(* IEC 61131-3 sources: SmartHomeNew/snapshots/2026-04-23, 16 files *)

(* ---- ST_Gateway_Command.dut ---- *)
{attribute 'pack_mode' := '1'}
TYPE ST_Gateway_Command :
STRUCT
    command_id : UDINT;
    timestamp_ms : UDINT;
    operator_id : STRING(10);
    command_type : E_Gateway_Command_Type;
    target_zone : BYTE;
    target_value : REAL;
    target_on_off : BOOL;
    target_scenario : E_SCENARIO_TYPE;
    target_armed : BOOL;
    target_pin : STRING(4);
    target_2fa_code : STRING(6);
    telegram_msg : STRING(200);
    source_ip : STRING(15); // IP-адрес источника команды для проверки безопасности
    crc32 : DWORD;
END_STRUCT
END_TYPE

(* ---- ST_Scenario_Config.dut ---- *)
{attribute 'pack_mode' := '1'}
TYPE ST_Scenario_Config :
STRUCT
    scenario_id : E_SCENARIO_TYPE;
    lighting_level_base : BYTE := 100;
    lighting_level_accent : BYTE := 100;
    floor_heating_adjust_celsius : REAL := 0.0;
    ventilation_speed_percent : BYTE := 50;
    sockets_enabled : BOOL := TRUE;
    blinds_position_percent : BYTE := 0;
    Presence_Simulation_Enabled : BOOL := FALSE;
END_STRUCT
END_TYPE

(* ---- ST_User_Rule.dut ---- *)
{attribute 'pack_mode' := '1'}
TYPE ST_User_Rule :
STRUCT
    Enabled : BOOL;
    Condition_Type : E_Rule_Condition_Type;
    Condition_Target_ID : BYTE; // ID зоны или датчика
    Condition_Op : E_Rule_Comparison;
    Condition_Value : REAL;
    Condition_Value_Max : REAL; // Для COMP_IN_RANGE
    Action_Target_ID : BYTE;
    Action_Value : REAL;
    Action_Type : E_Rule_Action_Type;
    Priority : BYTE;
END_STRUCT
END_TYPE

(* ---- GVL_CONFIG.gvl ---- *)
{attribute 'qualified_only'}
VAR_GLOBAL
    // Subsystem Configurations
    G_Heating_Config : ST_Heating_Config; // Настройки системы отопления
    G_Ventilation_Config : ST_Ventilation_Config; // Настройки системы вентиляции
    G_DHW_Config : ST_DHW_Config; // Настройки горячего водоснабжения
    G_Security_Config : ST_Security_Global_Config; // Настройки системы безопасности
    G_Flood_Config : ST_Flood_Config; // Настройки системы защиты от протечек

    // HMI Configurations
    G_HMI_FloorHeating_Configs : ARRAY[1..8] OF ST_FloorHeating_Circuit_Config; // Конфигурации контуров теплого пола
    G_Wet_Zone_Map : ARRAY[1..32] OF BOOL; // Карта мокрых зон (TRUE = мокрая зона)
    G_HMI_Tariff_Settings : ST_Tariff_Config; // Настройки тарифов
    G_HMI_Vent_Global_Config : ST_Ventilation_Global_Config; // Глобальные настройки вентиляции
    G_HMI_Vent_Unit_Configs : ARRAY[1..GVL_CONSTANTS.C_MAX_VENT_UNITS] OF ST_Ventilation_Unit_Config; // Конфигурации отдельных вентустановок
    G_HMI_Scenario_Configs : ARRAY[1..GVL_CONSTANTS.C_MAX_SCENARIOS] OF ST_Scenario_Config; // Конфигурации сценариев
    G_HMI_Outdoor_Configs : ARRAY[1..GVL_CONSTANTS.C_MAX_OUTDOOR_ZONES] OF ST_Outdoor_Zone_Config; // Конфигурации зон уличного освещения
    G_HMI_Flood_Config : ST_Flood_Global_Config; // Глобальные настройки защиты от протечек
    G_HMI_Gas_Config : ST_Gas_Valve_Configuration; // Конфигурация системы газового контроля
    G_HMI_Sensor_Calibrations : ARRAY[1..GVL_CONSTANTS.C_MAX_CALIBRATIONS] OF ST_Sensor_Calibration_Record; // Данные калибровки датчиков
    G_HMI_User_Rules : ARRAY[1..GVL_CONSTANTS.C_MAX_RULES] OF ST_User_Rule; // Пользовательские правила (Rule Engine)

    // Sensor calibration pipeline
    G_Enable_Sensor_Calibration : BOOL := TRUE;
    G_Calib_Outdoor_Temp : ST_Sensor_Calibration_Record;
    G_Calib_Supply_Temps : ARRAY[1..GVL_CONSTANTS.C_MAX_SUPPLY_TEMPS] OF ST_Sensor_Calibration_Record;
    G_Calib_Room_Temps : ARRAY[1..GVL_CONSTANTS.C_MAX_ZONES] OF ST_Sensor_Calibration_Record;
    G_Calib_Floor_Temps : ARRAY[1..GVL_CONSTANTS.C_MAX_ZONES] OF ST_Sensor_Calibration_Record;
    G_Calib_CO2 : ARRAY[1..GVL_CONSTANTS.C_MAX_ZONES] OF ST_Sensor_Calibration_Record;
    G_Calib_Humidity : ARRAY[1..GVL_CONSTANTS.C_MAX_ZONES] OF ST_Sensor_Calibration_Record;
    G_Calib_Manifold_T_Supply : ARRAY[1..GVL_CONSTANTS.C_MAX_MANIFOLDS] OF ST_Sensor_Calibration_Record;
    G_Calib_Manifold_T_Return : ARRAY[1..GVL_CONSTANTS.C_MAX_MANIFOLDS] OF ST_Sensor_Calibration_Record;
    G_Calib_Methane : ARRAY[1..GVL_CONSTANTS.C_MAX_METHANE_SENSORS] OF ST_Sensor_Calibration_Record;
    G_Calib_CO : ARRAY[1..GVL_CONSTANTS.C_MAX_CO_SENSORS] OF ST_Sensor_Calibration_Record;

    // Конфигурация тестирования клапанов
    G_Valve_Test_Config : ARRAY[1..GVL_CONSTANTS.C_MAX_MANIFOLDS] OF ST_Valve_Test_Config;

    // HMI Commands & States
    G_HMI_Cleaning_Mode_Active : ARRAY[1..GVL_CONSTANTS.C_MAX_CLEANING_MODES] OF BOOL; // Режим уборки активен
    G_HMI_Cleaning_Mode_TimeLeft : ARRAY[1..GVL_CONSTANTS.C_MAX_CLEANING_MODES] OF UINT; // Оставшееся время режима уборки
    G_HMI_Admin_2FA_Enabled : BOOL := FALSE; // Включена ли 2FA для ADMIN
    G_HMI_Current_Operator_Factor2_Done : BOOL; // Второй фактор пройден
    G_HMI_Current_Operator_ID : STRING(10); // ID текущего оператора
    G_HMI_Manual_Gas_Valve_Open : BOOL; // Ручное открытие газового клапана
    G_HMI_Manual_Gas_Valve_Time : UDINT := 5; // Время ручного открытия
    G_HMI_Manual_Gas_Valve_TimeLeft : UDINT; // Оставшееся время ручного открытия
    G_HMI_Apply_Settings : BOOL; // Команда: Применить настройки
    G_HMI_Mute_Alarm : BOOL; // Команда: Временное отключение сирены
    G_HMI_Ack_Alarms : BOOL; // Команда: Квитировать все тревоги

    // Access Control Commands
    G_HMI_Gate_Open_Req : BOOL; // Запрос на открытие въездных ворот
    G_HMI_Wicket_Open_Req : BOOL; // Запрос на открытие калитки
    G_HMI_Lock_1_Open_Req : BOOL; // Разблокировка основного замка
    G_HMI_Lock_1_Close_Req : BOOL; // Блокировка основного замка
    G_HMI_Lock_2_Open_Req : BOOL; // Разблокировка доп. замка
    G_HMI_Lock_2_Close_Req : BOOL; // Блокировка доп. замка

    // HMI Settings
    G_HMI_Language : BYTE := 0; // 0=RU, 1=EN
    G_HMI_Brightness : BYTE := 80;
    G_HMI_Screen_Saver_Timeout : UDINT := 300; // сек

    // Сетевая безопасность
    G_Allowed_IPs : ARRAY[1..GVL_CONSTANTS.C_MAX_ALLOWED_IPS] OF STRING(15) := ['192.168.1.100','192.168.1.101','127.0.0.1','','']; // Разрешенные IP-адреса для шлюза

    G_Backup_Circulation_Pump_In_Service : BOOL := TRUE; // Резервный насос доступен для логики
    G_Electric_Heater_In_Service : BOOL := TRUE; // Электронагреватель доступен для логики
    G_Freeze_Hardware_Retry_Count : INT := 2; // Количество повторных попыток для anti-freeze hardware
    G_Freeze_Hardware_Retry_Delay_MS : UDINT := 5000; // Задержка между попытками повторного пуска
    G_Pump_Exercise_Enabled : BOOL := TRUE; // Разрешение периодической прокрутки насосов после простоя
    G_Pump_Exercise_Interval_MS : UDINT := 604800000; // 7 суток
    G_Pump_Exercise_Duration_MS : UDINT := 30000; // 30 сек
    G_Manifold_Pump_In_Service : ARRAY[1..GVL_CONSTANTS.C_MAX_MANIFOLDS] OF BOOL := [TRUE, TRUE, TRUE, TRUE, TRUE];
    G_Manifold_Priority : ARRAY[1..GVL_CONSTANTS.C_MAX_MANIFOLDS] OF INT := [3, 3, 2, 2, 1]; // 3=high, 2=normal, 1=low
    G_Max_Active_Manifolds : INT := 3; // energy-management limit for simultaneous active manifolds
    G_Max_Thermal_Budget : REAL := 6.0; // simplified manifold thermal budget units
    G_DHW_Heating_Pump_In_Service : BOOL := TRUE;
    G_DHW_Circ_Pump_In_Service : BOOL := TRUE;
    G_Water_Valve_Exercise_Enabled : BOOL := TRUE;
    G_Water_Valve_Exercise_Interval_MS : UDINT := 604800000;
    G_Water_Valve_Exercise_Duration_MS : UDINT := 15000;
    G_Water_Valve_Exercise_Window_Start : TOD := TOD#04:00;
    G_Water_Valve_Exercise_Window_End : TOD := TOD#05:00;
    G_Water_Valve_Close_Retry_Count : INT := 2;
    G_Water_Valve_Close_Retry_Delay_MS : UDINT := 3000;
    // IO Mapping
    G_FloorTemp_Map : ARRAY[1..8] OF INT := [1, 2, 3, 4, 5, 6, 7, 8];
    G_RoomTemp_Map : ARRAY[1..16] OF INT := [1, 2, 3, 4, 5, 6, 7, 8, 9, 10, 11, 12, 13, 14, 15, 16];
    G_Door_Map : ARRAY[1..GVL_CONSTANTS.C_MAX_DOOR_SENSORS] OF INT := [1, 2, 3, 4, 5, 6, 7, 8];
    G_Window_Map : ARRAY[1..16] OF INT := [9, 10, 11, 12, 13, 14, 15, 16, 17, 18, 19, 20, 21, 22, 23, 24];

    // Evacuation config
    C_MAX_LIGHT_ZONES : INT := 32; // fallback if not defined elsewhere
    G_Evac_Exit_Zones : ARRAY[1..32] OF BOOL; // зоны-выходы (TRUE = выход)
    G_Evac_Smoke_Zone_Map : ARRAY[1..GVL_CONSTANTS.C_MAX_SMOKE_SENSORS] OF INT; // Привязка дымовых датчиков к зонам эвакуации
    G_Evac_Leak_Zone_Map : ARRAY[1..GVL_CONSTANTS.C_MAX_FLOOD_SENSORS] OF INT; // Привязка датчиков протечки к зонам эвакуации
    G_Evac_Gas_Zone_Map : ARRAY[1..GVL_CONSTANTS.C_MAX_METHANE_SENSORS] OF INT; // Привязка газовых датчиков к зонам эвакуации
    G_Evac_Zone_Names : ARRAY[1..32] OF STRING(80); // Человекочитаемые имена зон (помещения/крыло/этаж/сторона)

END_VAR

VAR_GLOBAL CONSTANT
    C_MS_PER_SEC    : UDINT := GVL_CONSTANTS.C_MS_IN_SECOND; // Миллисекунд в секунде
    C_SEC_PER_MIN   : UDINT := 60; // Секунд в минуте
    C_MIN_PER_HOUR  : UDINT := 60; // Минут в часе
    C_MS_PER_MIN    : UDINT := GVL_CONSTANTS.C_MS_IN_MINUTE; // Миллисекунд в минуте
    C_MAX_RULES     : INT := 20; // Максимальное количество пользовательских правил
    C_ZONE_COUNT    : BYTE := 18; // Общее количество зон в системе

    // Коды ошибок
    ERR_PRESSURE_OUT_OF_RANGE : UDINT := 16#E004;
    ERR_HIGH_DELTA_T : UDINT := 16#E005;
    ERR_BOILER_OFFLINE : UDINT := 16#E006;
    ERR_BOILER_GENERAL_FAULT : UDINT := 16#E007;
    ERR_BOILER_NO_FLAME : UDINT := 16#E008;
    ERR_PUMP_NO_CURRENT : UDINT := 16#E009;
    ERR_PUMP_UNDERCURRENT : UDINT := 16#E00A;
    ERR_PUMP_OVERCURRENT : UDINT := 16#E00B;
    ERR_DELTA_T_LOW : UDINT := 16#E00C;
    ERR_DELTA_T_HIGH : UDINT := 16#E00D;
    ERR_DHW_IO_OFFLINE : UDINT := 16#E00E;
    ERR_DHW_TEMP_SENSOR_FAULT : UDINT := 16#E00F;
    ERR_DHW_PRESSURE_OUT_OF_RANGE : UDINT := 16#E010;
    ERR_DHW_PRESSURE_SENSOR_FAULT : UDINT := 16#E011;
END_VAR

(* ---- GVL_IO.gvl ---- *)
{attribute 'qualified_only'}
VAR_GLOBAL
    DI_Security_Open : ARRAY[1..GVL_CONSTANTS.C_MAX_SECURITY_SENSORS] OF BOOL; // Дискретные входы: Герконы (нормально-замкнутые контакты, TRUE = Открыто)
    DI_Security_Glass : ARRAY[1..GVL_CONSTANTS.C_MAX_SECURITY_SENSORS] OF BOOL; // Дискретные входы: Датчики разбития стекла (активный уровень - TRUE)
    DI_Security_2F_Group : BOOL; // Дискретный вход: Групповой шлейф безопасности 2-го этажа (общий сигнал)
    DI_Flood_Sensors : ARRAY[1..GVL_CONSTANTS.C_MAX_FLOOD_SENSORS] OF BOOL; // Дискретные входы: Датчики протечки воды (активный уровень - TRUE)
    DI_Manifold_End_Switches : ARRAY[1..GVL_CONSTANTS.C_MAX_MANIFOLDS] OF BOOL; // Дискретные входы: Концевые выключатели клапанов коллекторов
    AO_Manifold_Valves : ARRAY[1..GVL_CONSTANTS.C_MAX_MANIFOLDS] OF UINT; // Аналоговые выходы: Приводы клапанов (0-10В, 0-1000 ед. для Modbus)
    DO_Manifold_Pumps : ARRAY[1..GVL_CONSTANTS.C_MAX_MANIFOLDS] OF BOOL; // Дискретные выходы: Циркуляционные насосы коллекторных узлов (220В)
    AI_Manifold_Currents : ARRAY[1..GVL_CONSTANTS.C_MAX_MANIFOLDS] OF INT; // Аналоговые входы: Обратная связь по току потребления насосов (диагностика)
    AI_Manifold_Pressures : ARRAY[1..GVL_CONSTANTS.C_MAX_MANIFOLDS] OF INT; // Аналоговые входы: Давление теплоносителя в коллекторах (0-10 бар)
    AI_Manifold_Temps_Supply : ARRAY[1..GVL_CONSTANTS.C_MAX_MANIFOLDS] OF ST_Owen_Analog_Value; // Аналоговые входы: Температура подачи (структура со статусом)
    AI_Manifold_Temps_Return : ARRAY[1..GVL_CONSTANTS.C_MAX_MANIFOLDS] OF INT; // Аналоговые входы: Температура обратной линии (в 10-х долях градуса)
    AO_Supply_Fans : ARRAY[1..GVL_CONSTANTS.C_MAX_SUPPLY_FANS] OF UINT; // Аналоговые выходы: Скорость приточных вентиляторов (0-10В)
    AO_Exhaust_Fans : ARRAY[1..GVL_CONSTANTS.C_MAX_EXHAUST_FANS] OF UINT; // Аналоговые выходы: Скорость вытяжных вентиляторов (0-10В)
    AO_Lighting_Levels : ARRAY[1..GVL_CONSTANTS.C_MAX_ZONES] OF UINT; // Аналоговые выходы: диммирование освещения (0-1000 -> 0..100%)
    AO_Blinds_Positions : ARRAY[1..GVL_CONSTANTS.C_MAX_BLINDS] OF UINT; // Аналоговые выходы: позиционирование штор/жалюзи (0-1000 -> 0..100%)
    AI_Supply_Temps : ARRAY[1..GVL_CONSTANTS.C_MAX_SUPPLY_TEMPS] OF ST_Owen_Analog_Value; // Аналоговые входы: Температура приточного воздуха после калорифера
    AI_Boiler_Modulation : ARRAY[1..GVL_CONSTANTS.C_MAX_BOILERS] OF INT; // Аналоговые входы: Текущий уровень модуляции мощности котла (%)
    AI_Boiler_Flame_Status : ARRAY[1..GVL_CONSTANTS.C_MAX_BOILERS] OF BOOL; // Дискретные входы: Датчик ионизации (подтверждение наличия пламени)
    DI_Boiler_Error : ARRAY[1..GVL_CONSTANTS.C_MAX_BOILERS] OF BOOL; // Дискретные входы: Сигнал общей ошибки/аварии котла
    AI_Methane_LEL : ARRAY[1..GVL_CONSTANTS.C_MAX_METHANE_SENSORS] OF ST_Owen_Analog_Value; // Аналоговые входы: Уровень метана CH4 (0-100% LEL)
    AI_CO_PPM : ARRAY[1..GVL_CONSTANTS.C_MAX_CO_SENSORS] OF REAL; // Аналоговые входы: Уровень угарного газа CO (PPM)
    DI_Smoke_Sensors : ARRAY[1..GVL_CONSTANTS.C_MAX_SMOKE_SENSORS] OF BOOL; // Дискретные входы: Оптические датчики дыма (пожарный шлейф)
    AI_Temp_Outdoor : ST_Owen_Analog_Value; // Аналоговый вход: Наружная температура воздуха (уличный датчик)
    AI_Floor_Temps : ARRAY[1..GVL_CONSTANTS.C_MAX_ZONES] OF REAL; // Аналоговые входы: Температура стяжки пола по зонам (датчики в гильзах)
    AI_Room_Temps : ARRAY[1..GVL_CONSTANTS.C_MAX_ZONES] OF REAL; // Аналоговые входы: Температура воздуха в помещениях (настенные датчики)
    AI_Room_Hum : ARRAY[1..GVL_CONSTANTS.C_MAX_ZONES] OF REAL; // Аналоговые входы: Влажность воздуха в помещениях (%)
    AI_Room_CO2 : ARRAY[1..GVL_CONSTANTS.C_MAX_ZONES] OF REAL; // Аналоговые входы: Уровень CO2 в помещениях (ppm)
    DO_Zone_Valves : ARRAY[1..GVL_CONSTANTS.C_MAX_ZONES] OF BOOL; // Дискретные выходы: Термоэлектрические приводы контуров (220В)
    AI_DHW_Temp : REAL; // Аналоговый вход: Температура воды в бойлере косвенного нагрева
    AI_DHW_Pressure : REAL; // Аналоговый вход: Давление в контуре ГВС (контроль подпитки и утечек)
    DO_DHW_Heating_Pump : BOOL; // Дискретный выход: Насос загрузки бойлера (первичный контур от котла)
    DO_DHW_Circ_Pump : BOOL; // Дискретный выход: Насос рециркуляции ГВС (кольцо потребителей)
    DO_Backup_Circulation_Pump : BOOL; // Дискретный выход: Резервный циркуляционный насос антизамерзания
    DO_Electric_Heater_Enable : BOOL; // Дискретный выход: Сухой контакт электрического нагревателя антизамерзания
    DI_Lighting_Switches : ARRAY[1..GVL_CONSTANTS.C_MAX_ZONES] OF BOOL; // Дискретные входы: Физические кнопки/выключатели (импульсные)
    DI_Socket_Switches : ARRAY[1..GVL_CONSTANTS.C_MAX_SOCKETS] OF BOOL; // Legacy-вход: локальные выключатели розеток отключены концептуально
    DI_Motion_Sensors : ARRAY[1..GVL_CONSTANTS.C_MAX_ZONES] OF BOOL; // Дискретные входы: Датчики присутствия (PIR-сенсоры)
    DO_Sockets : ARRAY[1..GVL_CONSTANTS.C_MAX_SOCKETS] OF BOOL; // Дискретные выходы: Управление розетками (реле)
    DO_Gas_Valve_Close : BOOL; // Дискретный выход: Импульс на закрытие электромагнитного газового клапана
    DO_Water_Valve_35_Close : BOOL; // Дискретный выход: Закрыть вводной шаровый кран воды №1 (с электроприводом)
    DO_Water_Valve_36_Close : BOOL; // Дискретный выход: Закрыть вводной шаровый кран воды №2 (с электроприводом)
    AI_Water_Valve_35_Current : REAL; // Аналоговый вход: Ток потребления электропривода крана №1 (контроль заклинивания)
    AI_Water_Valve_36_Current : REAL; // Аналоговый вход: Ток потребления электропривода крана №2 (контроль заклинивания)
    DI_Power_OK : BOOL; // Дискретный вход: Контроль наличия напряжения на вводе (реле контроля фаз)
    DO_Gas_Siren : BOOL; // Дискретный выход: Звуковое оповещение при опасной концентрации газа
    DO_Fire_Siren : BOOL; // Дискретный выход: Звуковое оповещение при обнаружении задымления
    DO_Security_Siren : BOOL; // Дискретный выход: Сирена охранной сигнализации
    DO_Pump_Main_Enable : BOOL; // Дискретный выход: Разрешение работы главного циркуляционного насоса системы
    DO_Gate_Open : BOOL; // Дискретный выход: Команда на открытие въездных ворот (импульс)
    DO_Wicket_Open : BOOL; // Дискретный выход: Команда на разблокировку электрозамка калитки
    DO_Lock_1_Open : BOOL; // Дискретный выход: Разблокировать основной электромеханический замок дома
    DO_Lock_1_Close : BOOL; // Дискретный выход: Заблокировать основной электромеханический замок дома
    DO_Lock_2_Open : BOOL; // Дискретный выход: Разблокировать дополнительный замок (черный ход)
    DO_Lock_2_Close : BOOL; // Дискретный выход: Заблокировать дополнительный замок (черный ход)
    DI_Partner_Pulse : BOOL; // Дискретный вход: Пульс от второго ПЛК
    DI_Partner_Active : BOOL; // Дискретный вход: Статус активности второго ПЛК
    DO_Heartbeat_Pulse : BOOL; // Дискретный выход: Собственный пульс
    DO_Active_Status : BOOL; // Дискретный выход: Собственный статус активности

    // Диагностика модулей ввода-вывода
    DI_Module_1_Heartbeat : BOOL; // Сигнал жизни от модуля 1
    DI_Module_2_Heartbeat : BOOL; // Сигнал жизни от модуля 2
    DI_Backup_Circulation_Pump_Feedback : BOOL; // Обратная связь резервного циркуляционного насоса
    DI_Electric_Heater_Feedback : BOOL; // Обратная связь электрического нагревателя
    DI_Water_Zone_Open_FB : ARRAY[1..32] OF BOOL; // Концевики: зональный водяной клапан открыт
    DI_Water_Zone_Close_FB : ARRAY[1..32] OF BOOL; // Концевики: зональный водяной клапан закрыт
    DO_Water_Zone_Enable : ARRAY[1..32] OF BOOL; // Разрешение подачи воды по зонам
END_VAR

(* ---- GVL_STATUS.gvl ---- *)
{attribute 'qualified_only'}
VAR_GLOBAL
    G_System_Time_MS : UDINT; // Системное время в миллисекундах
    G_Last_System_Time_MS : UDINT := 0; // Предыдущее системное время (для детекции переполнения)
    G_Time_Of_Day_MS : UDINT := 0; // Время от начала суток в мс (0-86399999)
    G_Current_Day : UINT := 1; // Текущий день недели (1-7)
    G_Day_Of_Year : UINT := 1; // Текущий день года (1-365)
    G_Current_TOD : TOD; // Текущее время суток
    G_Current_Scenario : E_SCENARIO_TYPE := E_SCENARIO_TYPE.SCENARIO_NONE; // Текущий активный сценарий
    G_Previous_Scenario : E_SCENARIO_TYPE := E_SCENARIO_TYPE.SCENARIO_NONE; // Предыдущий сценарий
    G_Is_Night : BOOL; // Флаг ночного времени
    G_PLC_ID : BYTE := 1; // 1 = PLC_A, 2 = PLC_B
    G_Is_Active_PLC : BOOL;
    G_Local_PLC_ID : BYTE := 1; // Идентификатор данного ПЛК в паре
    G_Active_PLC_ID : BYTE := 1; // Идентификатор ведущего ПЛК
    G_Remote_PLC_Pulse : BOOL; // Сигнал "жизни" от второго ПЛК
    G_Security_Status_Msg : STRING(200);
    G_Gas_Status_Msg : STRING(200);
    G_Flood_Status_Msg : STRING(200);
    G_Vent_Status_Msg : STRING(200);
    G_DHW_Status : ST_DHW_Status;
    G_Manifold_Status : ARRAY[1..GVL_CONSTANTS.C_MAX_MANIFOLDS] OF ST_Manifold_Status;
    G_Boiler_Status : ARRAY[1..GVL_CONSTANTS.C_MAX_BOILERS] OF ST_Boiler_Status;
    G_IO_Modules_Online : ARRAY[1..GVL_CONSTANTS.C_MAX_MODULES] OF BOOL; // Статусы модулей ввода-вывода
    G_Sim_Active : BOOL;
    G_Wet_Zone_Light_Active : BOOL;
    G_System_Mode_Msg : STRING(200); // Пояснение текущего режима работы системы для HMI
    G_System_Mode_Cause : STRING(200); // Корневая причина режима (пожар/газ/протечка/штатно)
    G_Evac_Target_Zone_Name : STRING(80); // Предпочтительная зона выхода/направления эвакуации
    G_Evac_Hazard_Zone_Name : STRING(80); // Наиболее важная опасная зона для HMI/диагностики
    G_Diagnostics : ST_System_Diagnostics; // Интегральная диагностика и HMI-состояния
END_VAR

(* ---- FB_Access_Control.st ---- *)
FUNCTION_BLOCK FB_Access_Control
VAR_INPUT
    VI_System_Time_MS   : UDINT; // Системное время (мс)
    VI_IsActivePLC      : BOOL; // Флаг: Данный ПЛК является ведущим (Active)
    VI_Armed            : BOOL; // Статус: Система безопасности находится под охраной
    VI_System_Mode      : E_System_Operating_Mode; // Агрегированный режим работы системы

    // Команды управления от HMI (через GVL_CONFIG)
    VI_Gate_Open_Req    : BOOL; // Запрос пользователя на открытие въездных ворот
    VI_Wicket_Open_Req  : BOOL; // Запрос пользователя на открытие калитки
    VI_Lock_1_Open_Req  : BOOL; // Запрос на разблокировку основного электрозамка дома
    VI_Lock_1_Close_Req : BOOL; // Запрос на блокировку основного электрозамка дома
    VI_Lock_2_Open_Req  : BOOL; // Запрос на разблокировку дополнительного электрозамка
    VI_Lock_2_Close_Req : BOOL; // Запрос на блокировку дополнительного электрозамка

    // Авторизация
    VI_PIN_Code         : STRING(4); // ПИН-код для авторизации
    VI_RFID_Tag         : STRING(20); // RFID/NFC метка для авторизации

    // Настройки из конфигурации безопасности (длительности импульсов)
    VI_Config           : ST_Security_Global_Config;
END_VAR
VAR_IN_OUT
    VI_Access_Codes     : ARRAY[1..GVL_CONSTANTS.C_MAX_ACCESS_CODES] OF DWORD;
    VI_RFID_Tags        : ARRAY[1..GVL_CONSTANTS.C_MAX_ACCESS_CODES] OF STRING(20);
END_VAR
VAR_OUTPUT
    VO_Gate_Open        : BOOL; // Выход: Импульс на открытие ворот (сухой контакт)
    VO_Wicket_Open      : BOOL; // Выход: Импульс на открытие калитки (электрозащелка)
    VO_Lock_1_Open      : BOOL; // Выход: Импульс на разблокировку замка №1
    VO_Lock_1_Close     : BOOL; // Выход: Импульс на блокировку замка №1
    VO_Lock_2_Open      : BOOL; // Выход: Импульс на разблокировку замка №2
    VO_Lock_2_Close     : BOOL; // Выход: Импульс на блокировку замка №2
END_VAR
VAR
    // Таймеры для формирования импульсов управления заданной длительности
    L_Gate_Timer        : TP; // Таймер импульса ворот
    L_Wicket_Timer      : TP; // Таймер импульса калитки
    L_Lock_1_Open_T     : TP; // Таймер открытия замка №1
    L_Lock_1_Close_T    : TP; // Таймер закрытия замка №1
    L_Lock_2_Open_T     : TP; // Таймер открытия замка №2
    L_Lock_2_Close_T    : TP; // Таймер закрытия замка №2

    L_Prev_Armed        : BOOL; // Предыдущее состояние охраны (для детекции фронта постановки)
    L_Auto_Lock_Req     : BOOL; // Флаг автоматического закрытия всех замков при постановке на охрану

    R_Trig_Gate         : R_TRIG;
    R_Trig_Wicket       : R_TRIG;
    R_Trig_Lock_1_O     : R_TRIG;
    R_Trig_Lock_1_C     : R_TRIG;
    R_Trig_Lock_2_O     : R_TRIG;
    R_Trig_Lock_2_C     : R_TRIG;

    fbAccessCode        : FB_AccessCode_Manager;
    L_Valid_PIN         : BOOL;
END_VAR

// Если ПЛК находится в режиме Standby (резерв), он не должен управлять выходами
IF NOT VI_IsActivePLC THEN
    RETURN;
END_IF;

IF VI_System_Mode = E_System_Operating_Mode.MODE_SAFE_STOP THEN
    VO_Gate_Open := FALSE;
    VO_Wicket_Open := FALSE;
    VO_Lock_1_Open := FALSE;
    VO_Lock_2_Open := FALSE;
    RETURN;
END_IF;

// 1. Логика автоматического закрытия замков при постановке на охрану (ТЗ 3.0)
// При переходе системы в режим "Охрана" принудительно блокируем все замки
IF VI_Armed AND NOT L_Prev_Armed THEN
    L_Auto_Lock_Req := TRUE;
END_IF;
L_Prev_Armed := VI_Armed;

// Детекторы фронта для команд
R_Trig_Gate(CLK := VI_Gate_Open_Req);
R_Trig_Wicket(CLK := VI_Wicket_Open_Req);
R_Trig_Lock_1_O(CLK := VI_Lock_1_Open_Req);
R_Trig_Lock_1_C(CLK := VI_Lock_1_Close_Req OR L_Auto_Lock_Req);
R_Trig_Lock_2_O(CLK := VI_Lock_2_Open_Req);
R_Trig_Lock_2_C(CLK := VI_Lock_2_Close_Req OR L_Auto_Lock_Req);

// Проверка PIN-кода или RFID-метки через менеджер кодов
fbAccessCode(
    VI_System_Time_MS := VI_System_Time_MS,
    VI_IsActivePLC := VI_IsActivePLC,
    VI_Code_To_Check := VI_PIN_Code,
    VI_RFID_To_Check := VI_RFID_Tag,
    VI_Access_Codes := VI_Access_Codes,
    VI_RFID_Tags := VI_RFID_Tags,
    VO_Code_Valid => L_Valid_PIN
);

// 2. Формирование импульсов управления исполнительными механизмами (Pulse Control)
// Открытие ворот и калитки требует валидного ПИН-кода или RFID-метки, если система под охраной
L_Gate_Timer(IN := R_Trig_Gate.Q AND (NOT VI_Armed OR L_Valid_PIN), PT := TO_TIME(VI_Config.gate_open_pulse_ms));
VO_Gate_Open := L_Gate_Timer.Q;

L_Wicket_Timer(IN := R_Trig_Wicket.Q AND (NOT VI_Armed OR L_Valid_PIN), PT := TO_TIME(VI_Config.wicket_open_pulse_ms));
VO_Wicket_Open := L_Wicket_Timer.Q;

L_Lock_1_Open_T(IN := R_Trig_Lock_1_O.Q AND (NOT VI_Armed OR L_Valid_PIN), PT := TO_TIME(VI_Config.lock_open_pulse_ms));
VO_Lock_1_Open := L_Lock_1_Open_T.Q;

L_Lock_1_Close_T(IN := R_Trig_Lock_1_C.Q, PT := TO_TIME(VI_Config.lock_close_pulse_ms));
VO_Lock_1_Close := L_Lock_1_Close_T.Q;

L_Lock_2_Open_T(IN := R_Trig_Lock_2_O.Q AND (NOT VI_Armed OR L_Valid_PIN), PT := TO_TIME(VI_Config.lock_open_pulse_ms));
VO_Lock_2_Open := L_Lock_2_Open_T.Q;

L_Lock_2_Close_T(IN := R_Trig_Lock_2_C.Q, PT := TO_TIME(VI_Config.lock_close_pulse_ms));
VO_Lock_2_Close := L_Lock_2_Close_T.Q;

// Сброс флага автоматического закрытия
IF L_Auto_Lock_Req THEN
    L_Auto_Lock_Req := FALSE;
END_IF;
// >>> BULK_SYNC_ANCHOR: FB_Access_Control <<<

(* ---- FB_AccessCode_Manager.st ---- *)
FUNCTION_BLOCK FB_AccessCode_Manager
VAR_INPUT
    VI_System_Time_MS : UDINT;
    VI_IsActivePLC    : BOOL;
    VI_Code_To_Check  : STRING(4);
    VI_RFID_To_Check  : STRING(20);
END_VAR
VAR_IN_OUT
    VI_Access_Codes   : ARRAY[1..GVL_CONSTANTS.C_MAX_ACCESS_CODES] OF DWORD;
    VI_RFID_Tags      : ARRAY[1..GVL_CONSTANTS.C_MAX_ACCESS_CODES] OF STRING(20);
END_VAR
VAR_OUTPUT
    VO_Code_Valid     : BOOL;
END_VAR
VAR
    L_i : INT;
    pCode : POINTER TO BYTE;
    L_CRC_Calc : FB_CRC32_Calculator;
    L_Input_Hash : DWORD;
END_VAR

VO_Code_Valid := FALSE;

// Вычисляем хэш введенного кода
IF LEN(VI_Code_To_Check) > 0 THEN
    pCode := ADR(VI_Code_To_Check);
    L_Input_Hash := 0;
    FOR L_i := 1 TO GVL_CONSTANTS.C_MAX_ACCESS_CODES DO
        IF VI_Access_Codes[L_i] <> 0 AND VI_Access_Codes[L_i] = L_Input_Hash THEN
            VO_Code_Valid := TRUE;
            RETURN;
        END_IF;
    END_FOR;
END_IF;

// Проверяем RFID метку
IF LEN(VI_RFID_To_Check) > 0 THEN
    FOR L_i := 1 TO GVL_CONSTANTS.C_MAX_ACCESS_CODES DO
        IF VI_RFID_Tags[L_i] <> '' AND VI_RFID_Tags[L_i] = VI_RFID_To_Check THEN
            VO_Code_Valid := TRUE;
            RETURN;
        END_IF;
    END_FOR;
END_IF;
// >>> BULK_SYNC_ANCHOR: FB_AccessCode_Manager <<<

(* ---- FB_Alarm_Manager.st ---- *)
FUNCTION_BLOCK FB_Alarm_Manager
VAR_INPUT
    VI_System_Time_MS : UDINT; // Системное время (мс)
    VI_IsActivePLC : BOOL; // Флаг: Данный ПЛК является ведущим

    // Входы от подсистем
    VI_Gas_Alarm : BOOL; // Сигнал тревоги: Утечка газа
    VI_Fire_Alarm : BOOL; // Сигнал тревоги: Пожар
    VI_Flood_Alarm : BOOL; // Сигнал тревоги: Протечка воды
    VI_Security_Alarm : BOOL; // Сигнал тревоги: Охранная система
    VI_First_Fault_Active : BOOL; // Активна защёлкнутая первая причина деградации
    VI_First_Fault_Type : INT; // 1=IO,2=Sensor,3=Comm,4=Subsystem
    VI_First_Fault_Source : INT; // 1=Heating,2=DHW,3=Ventilation,4=Lighting,5=Access

    // Сообщения от подсистем (для детализации)
    VI_Security_Msg : STRING(200); // Детальное сообщение от охранной системы

    // Команды с HMI
    VI_Acknowledge_All : BOOL; // Команда: Квитировать все тревоги
    VI_Mute_Siren : BOOL; // Команда: Временное отключение сирены
END_VAR
VAR_IN_OUT
    VI_Boiler_Errors : ARRAY[1..GVL_CONSTANTS.C_MAX_BOILERS] OF BOOL; // Ошибки котлов
END_VAR
VAR_IN_OUT
    VIO_Next_Alarm_ID : UDINT; // Глобальный счетчик ID тревог
END_VAR
VAR_OUTPUT
    VO_Global_Critical : BOOL; // Есть неквитированные критические аварии
    VO_Global_Warning : BOOL;  // Есть неквитированные предупреждения
    VO_Siren_Active : BOOL;    // Требуется включение сирены
    VO_Active_Count : INT;     // Количество активных тревог
    VO_Unacked_Count : INT;    // Количество неквитированных тревог
    VO_Event_Pulse : BOOL;     // Пульс события для History bridge
    VO_Event_Code : UDINT;     // 1201=ack all, 1202=alarm cleared, 1203=alarm created
    VO_Event_Value : REAL;     // Доп. значение события

    VO_Alarm_List : ARRAY[1..GVL_CONSTANTS.C_MAX_ALARMS] OF ST_Alarm_Record; // Список активных тревог для HMI
END_VAR
VAR
    L_i, L_j, L_k : INT;
    L_Target_Slot : INT;
    L_Min_Pri : INT;
    L_Pending_Alarms : ARRAY[1..10] OF ST_Alarm_Record;
    L_Pending_Count : INT := 0;

    // Фронты и антидребезг для детекции новых тревог
    T_Debounce_Gas : FB_System_Timer;
    T_Debounce_Fire : FB_System_Timer;
    T_Debounce_Flood : FB_System_Timer;
    T_Debounce_Security : FB_System_Timer;
    R_Trig_Gas : R_TRIG;
    R_Trig_Fire : R_TRIG;
    R_Trig_Flood : R_TRIG;
    R_Trig_Security : R_TRIG;
    R_Trig_First_Fault : R_TRIG;
    R_Trig_Boiler : ARRAY[1..GVL_CONSTANTS.C_MAX_BOILERS] OF R_TRIG;
    L_First_Fault_Source_Text : STRING(32);
    L_First_Fault_Type_Text : STRING(32);
    L_Event_Pulse_Latched : BOOL;
END_VAR

VO_Event_Pulse := FALSE;
VO_Event_Code := 0;
VO_Event_Value := 0.0;

// 1. Детекция новых тревог (антидребезг + передний фронт)
T_Debounce_Gas(IN := VI_Gas_Alarm, PT := T#100ms, VI_System_Time_MS := VI_System_Time_MS);
T_Debounce_Fire(IN := VI_Fire_Alarm, PT := T#100ms, VI_System_Time_MS := VI_System_Time_MS);
T_Debounce_Flood(IN := VI_Flood_Alarm, PT := T#500ms, VI_System_Time_MS := VI_System_Time_MS);
T_Debounce_Security(IN := VI_Security_Alarm, PT := T#100ms, VI_System_Time_MS := VI_System_Time_MS);

R_Trig_Gas(CLK := T_Debounce_Gas.Q);
R_Trig_Fire(CLK := T_Debounce_Fire.Q);
R_Trig_Flood(CLK := T_Debounce_Flood.Q);
R_Trig_Security(CLK := T_Debounce_Security.Q);
R_Trig_First_Fault(CLK := VI_First_Fault_Active);
FOR L_i := 1 TO GVL_CONSTANTS.C_MAX_BOILERS DO
    R_Trig_Boiler[L_i](CLK := VI_Boiler_Errors[L_i]);
END_FOR;

// 2. Добавление новых тревог в список (Кольцевой буфер)
L_Pending_Count := 0;
L_Event_Pulse_Latched := FALSE;

IF R_Trig_Gas.Q AND L_Pending_Count < 10 THEN
    L_Pending_Count := L_Pending_Count + 1;
    L_Pending_Alarms[L_Pending_Count].Timestamp_MS := VI_System_Time_MS;
    L_Pending_Alarms[L_Pending_Count].Source := 'Gas';
    L_Pending_Alarms[L_Pending_Count].Source_ID := 0;
    L_Pending_Alarms[L_Pending_Count].Message := 'Критическая концентрация газа!';
    L_Pending_Alarms[L_Pending_Count].Severity := E_ALERT_PRIORITY.ALERT_PRIORITY_CRITICAL;
    L_Pending_Alarms[L_Pending_Count].Is_Active := TRUE;
    L_Pending_Alarms[L_Pending_Count].Is_Acknowledged := FALSE;
END_IF;

IF R_Trig_Fire.Q AND L_Pending_Count < 10 THEN
    L_Pending_Count := L_Pending_Count + 1;
    L_Pending_Alarms[L_Pending_Count].Timestamp_MS := VI_System_Time_MS;
    L_Pending_Alarms[L_Pending_Count].Source := 'Fire';
    L_Pending_Alarms[L_Pending_Count].Source_ID := 0;
    L_Pending_Alarms[L_Pending_Count].Message := 'Обнаружено задымление!';
    L_Pending_Alarms[L_Pending_Count].Severity := E_ALERT_PRIORITY.ALERT_PRIORITY_CRITICAL;
    L_Pending_Alarms[L_Pending_Count].Is_Active := TRUE;
    L_Pending_Alarms[L_Pending_Count].Is_Acknowledged := FALSE;
END_IF;

IF R_Trig_Flood.Q AND L_Pending_Count < 10 THEN
    L_Pending_Count := L_Pending_Count + 1;
    L_Pending_Alarms[L_Pending_Count].Timestamp_MS := VI_System_Time_MS;
    L_Pending_Alarms[L_Pending_Count].Source := 'Flood';
    L_Pending_Alarms[L_Pending_Count].Source_ID := 0;
    L_Pending_Alarms[L_Pending_Count].Message := 'Обнаружена протечка воды!';
    L_Pending_Alarms[L_Pending_Count].Severity := E_ALERT_PRIORITY.ALERT_PRIORITY_CRITICAL;
    L_Pending_Alarms[L_Pending_Count].Is_Active := TRUE;
    L_Pending_Alarms[L_Pending_Count].Is_Acknowledged := FALSE;
END_IF;

IF R_Trig_Security.Q AND L_Pending_Count < 10 THEN
    L_Pending_Count := L_Pending_Count + 1;
    L_Pending_Alarms[L_Pending_Count].Timestamp_MS := VI_System_Time_MS;
    L_Pending_Alarms[L_Pending_Count].Source := 'Security';
    L_Pending_Alarms[L_Pending_Count].Source_ID := 0;
    L_Pending_Alarms[L_Pending_Count].Message := VI_Security_Msg;
    L_Pending_Alarms[L_Pending_Count].Severity := E_ALERT_PRIORITY.ALERT_PRIORITY_CRITICAL;
    L_Pending_Alarms[L_Pending_Count].Is_Active := TRUE;
    L_Pending_Alarms[L_Pending_Count].Is_Acknowledged := FALSE;
END_IF;

IF R_Trig_First_Fault.Q AND L_Pending_Count < 10 THEN
    L_Pending_Count := L_Pending_Count + 1;
    L_Pending_Alarms[L_Pending_Count].Timestamp_MS := VI_System_Time_MS;
    L_Pending_Alarms[L_Pending_Count].Source := 'Diagnostics';
    L_Pending_Alarms[L_Pending_Count].Source_ID := TO_BYTE(VI_First_Fault_Source);

    CASE VI_First_Fault_Type OF
        1: L_First_Fault_Type_Text := 'IO';
        2: L_First_Fault_Type_Text := 'Sensor';
        3: L_First_Fault_Type_Text := 'Comm';
        4: L_First_Fault_Type_Text := 'Subsystem';
        ELSE L_First_Fault_Type_Text := 'Unknown';
    END_CASE;

    CASE VI_First_Fault_Source OF
        1: L_First_Fault_Source_Text := 'Heating';
        2: L_First_Fault_Source_Text := 'DHW';
        3: L_First_Fault_Source_Text := 'Ventilation';
        4: L_First_Fault_Source_Text := 'Lighting';
        5: L_First_Fault_Source_Text := 'Access';
        ELSE L_First_Fault_Source_Text := 'Unknown';
    END_CASE;

    L_Pending_Alarms[L_Pending_Count].Message := CONCAT('Diagnostics root cause: ', CONCAT(L_First_Fault_Source_Text, CONCAT(' / ', L_First_Fault_Type_Text)));
    L_Pending_Alarms[L_Pending_Count].Severity := E_ALERT_PRIORITY.ALERT_PRIORITY_HIGH;
    L_Pending_Alarms[L_Pending_Count].Is_Active := TRUE;
    L_Pending_Alarms[L_Pending_Count].Is_Acknowledged := FALSE;
END_IF;

FOR L_j := 1 TO GVL_CONSTANTS.C_MAX_BOILERS DO
    IF R_Trig_Boiler[L_j].Q AND L_Pending_Count < 10 THEN
        L_Pending_Count := L_Pending_Count + 1;
        L_Pending_Alarms[L_Pending_Count].Timestamp_MS := VI_System_Time_MS;
        L_Pending_Alarms[L_Pending_Count].Source := 'Boiler';
        L_Pending_Alarms[L_Pending_Count].Source_ID := TO_BYTE(L_j);
        L_Pending_Alarms[L_Pending_Count].Message := CONCAT('Авария котла №', INT_TO_STRING(L_j));
        L_Pending_Alarms[L_Pending_Count].Severity := E_ALERT_PRIORITY.ALERT_PRIORITY_HIGH;
        L_Pending_Alarms[L_Pending_Count].Is_Active := TRUE;
        L_Pending_Alarms[L_Pending_Count].Is_Acknowledged := FALSE;
    END_IF;
END_FOR;

// Обработка очереди новых тревог с учетом приоритетов
FOR L_i := 1 TO L_Pending_Count DO

    L_Target_Slot := 0;

    // 1. Ищем пустой слот
    FOR L_k := 1 TO GVL_CONSTANTS.C_MAX_ALARMS DO
        IF VO_Alarm_List[L_k].ID = 0 THEN
            L_Target_Slot := L_k;
            EXIT;
        END_IF;
    END_FOR;

    // 2. Ищем квитированную тревогу с наименьшим приоритетом
    IF L_Target_Slot = 0 THEN
        L_Min_Pri := 999;
        FOR L_k := 1 TO GVL_CONSTANTS.C_MAX_ALARMS DO
            IF VO_Alarm_List[L_k].Is_Acknowledged AND TO_INT(VO_Alarm_List[L_k].Severity) < L_Min_Pri THEN
                L_Min_Pri := TO_INT(VO_Alarm_List[L_k].Severity);
                L_Target_Slot := L_k;
            END_IF;
        END_FOR;
    END_IF;

    // 3. Ищем неквитированную тревогу с наименьшим приоритетом (если он ниже добавляемой)
    IF L_Target_Slot = 0 THEN
        L_Min_Pri := 999;
        FOR L_k := 1 TO GVL_CONSTANTS.C_MAX_ALARMS DO
            IF TO_INT(VO_Alarm_List[L_k].Severity) < L_Min_Pri AND TO_INT(VO_Alarm_List[L_k].Severity) < TO_INT(L_Pending_Alarms[L_i].Severity) THEN
                L_Min_Pri := TO_INT(VO_Alarm_List[L_k].Severity);
                L_Target_Slot := L_k;
            END_IF;
        END_FOR;
    END_IF;

    IF L_Target_Slot = 0 THEN
        // Буфер полон критических неквитированных тревог. Не затираем!
        CONTINUE;
    END_IF;

    VO_Alarm_List[L_Target_Slot] := L_Pending_Alarms[L_i];
    VO_Alarm_List[L_Target_Slot].ID := VIO_Next_Alarm_ID;
    VIO_Next_Alarm_ID := VIO_Next_Alarm_ID + 1;
    IF VIO_Next_Alarm_ID = 0 THEN VIO_Next_Alarm_ID := 1; END_IF;
    IF NOT L_Event_Pulse_Latched THEN
        VO_Event_Pulse := TRUE;
        VO_Event_Code := 1203;
        VO_Event_Value := TO_REAL(VO_Alarm_List[L_Target_Slot].Severity);
        L_Event_Pulse_Latched := TRUE;
    END_IF;
END_FOR;

// 3. Обновление статуса существующих тревог (ушли ли они?)
FOR L_i := 1 TO GVL_CONSTANTS.C_MAX_ALARMS DO
    IF VO_Alarm_List[L_i].ID <> 0 THEN
        IF VO_Alarm_List[L_i].Source = 'Gas' THEN VO_Alarm_List[L_i].Is_Active := VI_Gas_Alarm;
        ELSIF VO_Alarm_List[L_i].Source = 'Fire' THEN VO_Alarm_List[L_i].Is_Active := VI_Fire_Alarm;
        ELSIF VO_Alarm_List[L_i].Source = 'Flood' THEN VO_Alarm_List[L_i].Is_Active := VI_Flood_Alarm;
        ELSIF VO_Alarm_List[L_i].Source = 'Security' THEN VO_Alarm_List[L_i].Is_Active := VI_Security_Alarm;
        ELSIF VO_Alarm_List[L_i].Source = 'Diagnostics' THEN VO_Alarm_List[L_i].Is_Active := VI_First_Fault_Active;
        ELSIF VO_Alarm_List[L_i].Source = 'Boiler' THEN
            IF TO_INT(VO_Alarm_List[L_i].Source_ID) >= 1 AND TO_INT(VO_Alarm_List[L_i].Source_ID) <= GVL_CONSTANTS.C_MAX_BOILERS THEN
                VO_Alarm_List[L_i].Is_Active := VI_Boiler_Errors[TO_INT(VO_Alarm_List[L_i].Source_ID)];
            END_IF;
        END_IF;
    END_IF;
END_FOR;

// 4. Квитирование тревог
IF VI_Acknowledge_All THEN
    FOR L_i := 1 TO GVL_CONSTANTS.C_MAX_ALARMS DO
        IF VO_Alarm_List[L_i].ID <> 0 THEN
            VO_Alarm_List[L_i].Is_Acknowledged := TRUE;
        END_IF;
    END_FOR;

    IF NOT L_Event_Pulse_Latched THEN
        VO_Event_Pulse := TRUE;
        VO_Event_Code := 1201;
        VO_Event_Value := TO_REAL(VO_Unacked_Count);
        L_Event_Pulse_Latched := TRUE;
    END_IF;
END_IF;

// 4.5 Автоквитирование некритичных тревог, если они больше не активны
FOR L_i := 1 TO GVL_CONSTANTS.C_MAX_ALARMS DO
    IF VO_Alarm_List[L_i].ID <> 0 AND NOT VO_Alarm_List[L_i].Is_Active AND NOT VO_Alarm_List[L_i].Is_Acknowledged THEN
        IF VO_Alarm_List[L_i].Severity <> E_ALERT_PRIORITY.ALERT_PRIORITY_CRITICAL THEN
            VO_Alarm_List[L_i].Is_Acknowledged := TRUE;
        END_IF;
    END_IF;
END_FOR;

// 5. Очистка списка (удаление неактивных И квитированных тревог)
// В кольцевом буфере мы просто помечаем слот как пустой (ID = 0), без сдвига массива
FOR L_i := 1 TO GVL_CONSTANTS.C_MAX_ALARMS DO
    IF VO_Alarm_List[L_i].ID <> 0 AND NOT VO_Alarm_List[L_i].Is_Active AND VO_Alarm_List[L_i].Is_Acknowledged THEN
        // Удаляем тревогу
        VO_Alarm_List[L_i].ID := 0;
        IF NOT L_Event_Pulse_Latched THEN
            VO_Event_Pulse := TRUE;
            VO_Event_Code := 1202;
            VO_Event_Value := 0.0;
            L_Event_Pulse_Latched := TRUE;
        END_IF;
    END_IF;
END_FOR;

// 6. Подсчет статистики и формирование глобальных флагов
VO_Global_Critical := FALSE;
VO_Global_Warning := FALSE;
VO_Siren_Active := FALSE;
VO_Active_Count := 0;
VO_Unacked_Count := 0;

FOR L_i := 1 TO GVL_CONSTANTS.C_MAX_ALARMS DO
    IF VO_Alarm_List[L_i].ID <> 0 THEN
        IF VO_Alarm_List[L_i].Is_Active THEN
            VO_Active_Count := VO_Active_Count + 1;
        END_IF;

        IF NOT VO_Alarm_List[L_i].Is_Acknowledged THEN
            VO_Unacked_Count := VO_Unacked_Count + 1;

            IF VO_Alarm_List[L_i].Severity = E_ALERT_PRIORITY.ALERT_PRIORITY_CRITICAL THEN
                VO_Global_Critical := TRUE;
                // Сирена работает только для неквитированных критических тревог, если не включен Mute
                IF NOT VI_Mute_Siren THEN
                    VO_Siren_Active := TRUE;
                END_IF;
            ELSIF VO_Alarm_List[L_i].Severity = E_ALERT_PRIORITY.ALERT_PRIORITY_HIGH THEN
                VO_Global_Warning := TRUE;
            END_IF;
        END_IF;
    END_IF;
END_FOR;
// >>> BULK_SYNC_ANCHOR: FB_Alarm_Manager <<<

(* ---- FB_Heating_System_Manager.st ---- *)
// ==============================================================================
// Блок управления системой отопления (Heating System Manager)
// Назначение:
// - Управление контурами теплого пола (открытие/закрытие клапанов).
// - Управление насосами коллекторов и смесительными узлами.
// - Управление каскадом котлов (ротация, расчет ресурса).
// - Защита от перегрева и замерзания.
// - Интеграция с Rule Engine.
// ==============================================================================
FUNCTION_BLOCK FB_Heating_System_Manager
VAR_INPUT
    VI_Preheat_Request : BOOL; // preheat scenario trigger
    L_Climate_Zone_ID : INT;

    VI_System_Mode : E_System_Operating_Mode; // System mode from State Manager

    VI_System_Time_MS : UDINT; // Системное время (мс)
    VI_Current_TOD : TOD; // Текущее время суток
    VI_IsActivePLC : BOOL; // Флаг: Данный ПЛК является ведущим
    VI_Outdoor_Temp : REAL; // Уличная температура воздуха (°C)
    VI_Config : ST_Heating_Config; // Конфигурация системы отопления
    VI_Tariff : ST_Tariff_Config; // Настройки тарифов
    VI_Current_Hour : UINT; // Текущий час (0-23)
    VI_Boiler_Stop : BOOL; // Команда на остановку котлов (от газовой/пожарной сигнализации); вход сохранён для совместимости, не используется как direct control
    VI_DHW_Heating_Demand : BOOL; // Запрос тепла от бойлера ГВС (приоритет)
    VI_DHW_Target_Temp : REAL; // Целевая температура бойлера ГВС
    VI_Current_Scenario : E_SCENARIO_TYPE; // Текущий сценарий
    VI_Emergency_Stop : BOOL; // Агрегированный аварийный стоп от подсистемы безопасности
    VI_Gas_Safety_Stop : BOOL; // Газовая авария / закрытие газового клапана
    VI_Boiler_Error_Status : ARRAY[1..GVL_CONSTANTS.C_MAX_BOILERS] OF BOOL; // Ошибки котлов / ошибка адаптера
    VI_Boiler_OT_Online : ARRAY[1..GVL_CONSTANTS.C_MAX_BOILERS] OF BOOL; // Признак доступности OpenTherm-канала
    VI_Boiler_Modulation : ARRAY[1..GVL_CONSTANTS.C_MAX_BOILERS] OF REAL; // Текущая модуляция котлов (%)
END_VAR
VAR_IN_OUT
    VI_Floor_Temps : ARRAY[1..8] OF REAL; // Температуры стяжки пола по зонам
    VI_Room_Temps : ARRAY[1..16] OF REAL; // Температуры воздуха в помещениях
    VI_Manifold_Pressures : ARRAY[1..GVL_CONSTANTS.C_MAX_MANIFOLDS] OF REAL; // Давление в коллекторах (бар)
    VI_Manifold_Currents : ARRAY[1..GVL_CONSTANTS.C_MAX_MANIFOLDS] OF REAL; // Ток насосов коллекторов (мА)
    VI_Manifold_Temps_Supply : ARRAY[1..GVL_CONSTANTS.C_MAX_MANIFOLDS] OF REAL; // Температура подачи на коллекторах
    VI_Manifold_Temps_Return : ARRAY[1..GVL_CONSTANTS.C_MAX_MANIFOLDS] OF REAL; // Температура обратки на коллекторах
    VI_Boiler_Flame_Status : ARRAY[1..GVL_CONSTANTS.C_MAX_BOILERS] OF BOOL; // Статус наличия пламени в котлах
    VI_Zone_Configs : ARRAY[1..8] OF ST_FloorHeating_Circuit_Config; // Конфигурации контуров
    VI_Rule_Actions : ARRAY[1..GVL_CONSTANTS.C_MAX_RULES] OF ST_Rule_Action; // Действия от Rule Engine
    VI_IO_Modules_Online : ARRAY[1..GVL_CONSTANTS.C_MAX_MODULES] OF BOOL; // Статусы модулей ввода-вывода
    VI_Scenario_Configs : ARRAY[1..GVL_CONSTANTS.C_MAX_SCENARIOS] OF ST_Scenario_Config; // Конфигурации сценариев
    VI_Manifold_End_Switches : ARRAY[1..GVL_CONSTANTS.C_MAX_MANIFOLDS] OF BOOL; // Концевики клапанов
    VI_Valve_Test_Config : ARRAY[1..GVL_CONSTANTS.C_MAX_MANIFOLDS] OF ST_Valve_Test_Config; // Конфигурация тестирования клапанов
END_VAR

VAR_OUTPUT
    VO_Manifold_Valves : ARRAY[1..GVL_CONSTANTS.C_MAX_MANIFOLDS] OF REAL; // Выход: Положение клапанов смесителей (0-100%)
    VO_Manifold_Pumps : ARRAY[1..GVL_CONSTANTS.C_MAX_MANIFOLDS] OF BOOL; // Выход: Управление насосами коллекторов
    VO_Zone_Valves : ARRAY[1..8] OF BOOL; // Выход: Управление клапанами контуров (Зоны 1-16)
    VO_Boiler_OT_Enable : ARRAY[1..GVL_CONSTANTS.C_MAX_BOILERS] OF BOOL; // Физические команды в OpenTherm
    VO_Boiler_OT_Setpoint : ARRAY[1..GVL_CONSTANTS.C_MAX_BOILERS] OF REAL; // Физические уставки в OpenTherm
    VO_Backup_Circulation_Pump : BOOL; // Резервный циркуляционный насос в режиме антизамерзания при газовой аварии
    VO_Electric_Heater_Enable : BOOL; // Сухой контакт электрического нагревателя антизамерзания
    VO_Freeze_Risk_Status : BOOL; // Признак риска замерзания при защёлкнутой газовой аварии
    VO_Status : ARRAY[1..GVL_CONSTANTS.C_MAX_MANIFOLDS] OF ST_Manifold_Status; // Сводный статус коллекторных узлов для HMI
    VO_Boiler_Status : ARRAY[1..GVL_CONSTANTS.C_MAX_BOILERS] OF ST_Boiler_Status; // Сводный статус котлов для HMI
END_VAR

VAR

    L_PID_Valves : ARRAY[1..GVL_CONSTANTS.C_MAX_MANIFOLDS] OF FB_PID_Controller; // ПИД-регуляторы для поддержания температуры подачи
    L_PID_Timer : ARRAY[1..GVL_CONSTANTS.C_MAX_MANIFOLDS] OF FB_System_Timer; // Таймеры вызова ПИД-регуляторов
    L_Floor_Controllers : ARRAY[1..8] OF FB_FloorHeating_Controller; // Контроллеры зон теплого пола
    L_Last_Boiler_Rotation : UDINT; // Время последней ротации ведущего котла
    L_Lead_Boiler : BYTE := 1; // Номер ведущего котла (1 или 2)
    L_i : INT; // Индекс для циклов
    L_Zone_Config : ST_FloorHeating_Circuit_Config;
    L_j : INT; // Вспомогательный индекс
    L_Target_Supply_Temp : REAL; // Рассчитанная целевая температура подачи
    L_Demand_Power : REAL; // Суммарный запрос мощности от всех коллекторов
    L_Any_Zone_Active : ARRAY[1..GVL_CONSTANTS.C_MAX_MANIFOLDS] OF BOOL; // Флаги наличия запроса тепла по коллекторам
    L_Current_Temp : REAL; // Текущая температура для ПИД
    L_Sensor_Error : BOOL; // Ошибка обоих датчиков

    // Плавный переход сценария
    L_Prev_Scenario : E_SCENARIO_TYPE;
    L_Scenario_Adjust : REAL;
    L_Target_Scenario_Adjust : REAL;
    L_Transition_Temp : FB_Scenario_Transition_Controller;

    // ТЗ 2.5: Защита от перегрева стяжки
    L_Overheat_Timer : ARRAY[1..8] OF FB_System_Timer; // Таймеры задержки отключения при перегреве

    // ТЗ 2.6: Сервисная диагностика и паузы
    L_Pump_Run_Timer : ARRAY[1..GVL_CONSTANTS.C_MAX_MANIFOLDS] OF FB_System_Timer; // Таймер непрерывной работы насоса (до 72ч)
    L_Pump_Pause_Timer : ARRAY[1..GVL_CONSTANTS.C_MAX_MANIFOLDS] OF FB_System_Timer; // Таймер обязательной паузы насоса (1ч)
    L_Pump_In_Pause : ARRAY[1..GVL_CONSTANTS.C_MAX_MANIFOLDS] OF BOOL; // Флаг: Насос находится в режиме сервисной паузы

    // ТЗ 2.8: Учет ресурса оборудования
    L_Last_Scan_Time : UDINT; // Время предыдущего цикла для расчета наработки
    L_Scan_Time_Init : BOOL := FALSE;
    L_Lifespan_S : REAL := 50000.0 * 3600.0; // Расчетный ресурс котла (50,000 часов в секундах)
    L_Delta_MS : UDINT; // Разница времени
    L_Pump_Diag : ARRAY[1..GVL_CONSTANTS.C_MAX_MANIFOLDS] OF FB_Device_Predictive_Diag; // Диагностика насосов
    L_Boiler_Life : ARRAY[1..GVL_CONSTANTS.C_MAX_BOILERS] OF FB_Lifetime_Predictor; // Предиктор ресурса котлов

    fbFloorTempValidator : ARRAY[1..8] OF FB_Analog_Validator;
    fbRoomTempValidator : ARRAY[1..16] OF FB_Analog_Validator;
    fbValveTestManager : FB_Valve_Test_Manager; // Менеджер тестирования клапанов
    fbBoilerCascade : FB_Boiler_Cascade_Manager; // Выделенный менеджер каскада котлов
    fbBoilerOpenTherm : FB_Boiler_OpenTherm_Interface; // Основной транспорт OpenTherm
    L_IO_Failsafe_Active : BOOL; // Флаг потери связи с модулями I/O
    L_Freeze_Mode_Active : BOOL; // Флаг антизамерзания по ТЗ
    L_Freeze_Target_Supply : REAL; // Уставка подачи в режиме антизамерзания
    L_Delta_T : REAL; // Разница температур подача/обратка
    L_Min_Supply_Temp : REAL; // Минимальная температура теплоносителя для антизамерзания
    L_Boiler_OT_Command_Valid : ARRAY[1..GVL_CONSTANTS.C_MAX_BOILERS] OF BOOL; // Команда ушла через OT
    L_Boiler_Request_Enable : ARRAY[1..GVL_CONSTANTS.C_MAX_BOILERS] OF BOOL; // Внутренний request на котлы от логики каскада
    L_Boiler_Request_Setpoint : ARRAY[1..GVL_CONSTANTS.C_MAX_BOILERS] OF REAL; // Внутренняя request-уставка котлов
    L_Policy_Normal : BOOL; // Policy: normal operation
    L_Policy_Safe_Stop : BOOL; // Policy: hard safe stop
    L_Policy_Degraded : BOOL; // Policy: limited conservative operation
    L_Policy_Freeze_Protection : BOOL; // Policy: freeze protection mode
    L_Any_Sensor_Error : BOOL;
    L_Any_Subsystem_Degraded : BOOL;
    L_Adaptive_Max_Delta : REAL;
    L_Adaptive_Delta : REAL;
    L_Adaptive_Zone_i : INT;
    L_Adaptive_Weighted_Sum : REAL;
    L_Adaptive_Weight_Total : REAL;
    L_Adaptive_Effective_Delta : REAL;
    L_Adaptive_Weight : REAL;
    L_Adaptive_Correction : REAL;
END_VAR

// ========================================
// Heating policy layer
// ========================================
L_Policy_Normal := (VI_System_Mode = E_System_Operating_Mode.MODE_NORMAL);
L_Policy_Safe_Stop := (VI_System_Mode = E_System_Operating_Mode.MODE_SAFE_STOP);
L_Policy_Degraded := (VI_System_Mode = E_System_Operating_Mode.MODE_DEGRADED);
L_Policy_Freeze_Protection := (VI_System_Mode = E_System_Operating_Mode.MODE_FREEZE_PROTECTION);

// ========================================
// Heating freeze policy activation
// ========================================
IF L_Policy_Freeze_Protection THEN
    L_Freeze_Mode_Active := TRUE;
END_IF;

// 0. Агрегация деградации для system mode
GVL_STATE.G_Heating_IO_Fault := FALSE;
GVL_STATE.G_Heating_Sensor_Fault := FALSE;
GVL_STATE.G_Heating_Subsystem_Degraded := FALSE;
L_Any_Sensor_Error := FALSE;
L_Any_Subsystem_Degraded := FALSE;

// 0. Аварийный стоп от подсистемы безопасности
VO_Backup_Circulation_Pump := FALSE;
VO_Electric_Heater_Enable := FALSE;
VO_Freeze_Risk_Status := FALSE;

IF VI_Gas_Safety_Stop THEN
    L_Freeze_Mode_Active := (VI_Outdoor_Temp < -5.0);
    FOR L_i := 1 TO GVL_CONSTANTS.C_MAX_HEATING_CIRCUITS DO
        IF VI_Floor_Temps[L_i] < 7.0 THEN
            L_Freeze_Mode_Active := TRUE;
        END_IF;
        VO_Zone_Valves[L_i] := FALSE;
    END_FOR;

    FOR L_i := 1 TO GVL_CONSTANTS.C_MAX_MANIFOLDS DO
        VO_Manifold_Pumps[L_i] := FALSE;
        VO_Manifold_Valves[L_i] := 0.0;
    END_FOR;

    FOR L_i := 1 TO GVL_CONSTANTS.C_MAX_BOILERS DO
        VO_Boiler_OT_Enable[L_i] := FALSE;
        VO_Boiler_OT_Setpoint[L_i] := 0.0;
        VO_Boiler_Status[L_i].Warning := FALSE;
        VO_Boiler_Status[L_i].Error := TRUE;
    END_FOR;

    IF L_Freeze_Mode_Active THEN
        VO_Backup_Circulation_Pump := TRUE;
        L_Freeze_Target_Supply := LIMIT(20.0, VI_Config.Freeze_Threshold + 2.0, 35.0);
        L_Min_Supply_Temp := 1000.0;
        FOR L_i := 1 TO GVL_CONSTANTS.C_MAX_MANIFOLDS DO
            IF VI_Manifold_Temps_Supply[L_i] < L_Min_Supply_Temp THEN
                L_Min_Supply_Temp := VI_Manifold_Temps_Supply[L_i];
            END_IF;
        END_FOR;
        IF L_Min_Supply_Temp > 900.0 THEN
            L_Min_Supply_Temp := 0.0;
        END_IF;

        IF L_Min_Supply_Temp < (L_Freeze_Target_Supply - 1.0) THEN
            VO_Electric_Heater_Enable := TRUE;
        ELSIF L_Min_Supply_Temp > (L_Freeze_Target_Supply + 1.0) THEN
            VO_Electric_Heater_Enable := FALSE;
        END_IF;

        // При защёлкнутой газовой аварии оператор должен видеть, что система живёт в деградированном anti-freeze режиме.
        VO_Freeze_Risk_Status := TRUE;
    END_IF;

    RETURN;
END_IF;

IF VI_Emergency_Stop OR L_Policy_Safe_Stop THEN
    FOR L_i := 1 TO GVL_CONSTANTS.C_MAX_HEATING_CIRCUITS DO
        VO_Zone_Valves[L_i] := FALSE;
    END_FOR;

    FOR L_i := 1 TO GVL_CONSTANTS.C_MAX_MANIFOLDS DO
        VO_Manifold_Pumps[L_i] := FALSE;
        VO_Manifold_Valves[L_i] := 0.0;
    END_FOR;

    FOR L_i := 1 TO GVL_CONSTANTS.C_MAX_BOILERS DO
        VO_Boiler_OT_Enable[L_i] := FALSE;
        VO_Boiler_OT_Setpoint[L_i] := 0.0;
        VO_Boiler_Status[L_i].Warning := FALSE;
        VO_Boiler_Status[L_i].Error := TRUE;
    END_FOR;

    RETURN;
END_IF;

// 1. Проверка связи с модулями ввода-вывода (ТЗ 2.0)
L_IO_Failsafe_Active := FALSE;
FOR L_i := 1 TO GVL_CONSTANTS.C_MAX_MODULES DO
    IF NOT VI_IO_Modules_Online[L_i] THEN
        L_IO_Failsafe_Active := TRUE;
        GVL_STATE.G_Heating_IO_Fault := TRUE;
GVL_STATE.G_Heating_Subsystem_Degraded := TRUE;
        EXIT;
    END_IF;
END_FOR;

IF L_IO_Failsafe_Active THEN
    // Fail-safe: закрываем зональные клапаны, чтобы не разгонять неконтролируемые контуры,
    // но при риске замерзания сохраняем минимальную циркуляцию и минимальную теплогенерацию.
    L_Freeze_Mode_Active := (VI_Outdoor_Temp < -5.0);

    FOR L_j := 1 TO GVL_CONSTANTS.C_MAX_HEATING_CIRCUITS DO
        IF VI_Floor_Temps[L_j] < 7.0 THEN
            L_Freeze_Mode_Active := TRUE;
        END_IF;
        VO_Zone_Valves[L_j] := FALSE;
    END_FOR;

    IF L_Freeze_Mode_Active THEN
        L_Freeze_Target_Supply := LIMIT(20.0, VI_Config.Freeze_Threshold + 2.0, 35.0);
    ELSE
        L_Freeze_Target_Supply := 0.0;
    END_IF;

    FOR L_j := 1 TO GVL_CONSTANTS.C_MAX_MANIFOLDS DO
        IF L_Freeze_Mode_Active THEN
            VO_Manifold_Pumps[L_j] := TRUE;
            VO_Manifold_Valves[L_j] := 35.0;
        ELSE
            VO_Manifold_Pumps[L_j] := FALSE;
            VO_Manifold_Valves[L_j] := 0.0;
        END_IF;
    END_FOR;

    // В аварийном I/O режиме напрямую формируем только legacy request-мirror.
    // Реальные физические команды всё равно будут интерпретированы transport-слоем выше по архитектуре.
    FOR L_j := 1 TO GVL_CONSTANTS.C_MAX_BOILERS DO
        VO_Boiler_OT_Enable[L_j] := FALSE;
        VO_Boiler_OT_Setpoint[L_j] := 0.0;
    END_FOR;

    IF L_Freeze_Mode_Active THEN
        // В fail-safe используем только ведущий аварийный вариант: котёл №1 на минимальной уставке.
        IF VI_Boiler_OT_Online[1] AND NOT VI_Boiler_Error_Status[1] THEN
            VO_Boiler_OT_Enable[1] := TRUE;
            VO_Boiler_OT_Setpoint[1] := L_Freeze_Target_Supply;
        END_IF;
    END_IF;

    RETURN;
END_IF;

// --- HEATING TARGET INJECTION ---
// Global arbitration target is applied after base policy calculation.
IF GVL_STATE.G_Target_Temperature > 0.0 THEN
    L_Target_Supply_Temp := GVL_STATE.G_Target_Temperature;
END_IF;

// --- MULTI-ZONE ADAPTIVE CORRECTION ---
// Final adaptive refinement layer.
L_Adaptive_Max_Delta := 0.0;
L_Adaptive_Weighted_Sum := 0.0;
L_Adaptive_Weight_Total := 0.0;
L_Adaptive_Effective_Delta := 0.0;
L_Adaptive_Correction := 0.0;

FOR L_Adaptive_Zone_i := 1 TO 8 DO
    IF VI_Zone_Configs[L_Adaptive_Zone_i].zone >= 1 AND VI_Zone_Configs[L_Adaptive_Zone_i].zone <= 8 THEN
        CASE VI_Zone_Configs[L_Adaptive_Zone_i].control_type OF
            0:
                L_Adaptive_Delta :=
                    VI_Zone_Configs[L_Adaptive_Zone_i].design_temp -
                    VI_Floor_Temps[L_Adaptive_Zone_i];
                L_Adaptive_Weight := 0.6;
            1, 2:
                L_Adaptive_Delta :=
                    VI_Zone_Configs[L_Adaptive_Zone_i].design_temp -
                    VI_Room_Temps[VI_Zone_Configs[L_Adaptive_Zone_i].zone];
                L_Adaptive_Weight := 1.0;
            ELSE
                L_Adaptive_Delta :=
                    VI_Zone_Configs[L_Adaptive_Zone_i].design_temp -
                    VI_Room_Temps[VI_Zone_Configs[L_Adaptive_Zone_i].zone];
                L_Adaptive_Weight := 0.8;
        END_CASE;

        IF VI_Zone_Configs[L_Adaptive_Zone_i].zone >= 1 AND VI_Zone_Configs[L_Adaptive_Zone_i].zone <= 4 THEN
            L_Adaptive_Weight := L_Adaptive_Weight * 1.2;
        ELSIF VI_Zone_Configs[L_Adaptive_Zone_i].zone >= 9 THEN
            L_Adaptive_Weight := L_Adaptive_Weight * 0.7;
        END_IF;

        IF L_Adaptive_Weight > 2.0 THEN
            L_Adaptive_Weight := 2.0;
        ELSIF L_Adaptive_Weight < 0.2 THEN
            L_Adaptive_Weight := 0.2;
        END_IF;

        IF L_Adaptive_Delta > L_Adaptive_Max_Delta THEN
            L_Adaptive_Max_Delta := L_Adaptive_Delta;
        END_IF;

        L_Adaptive_Weighted_Sum := L_Adaptive_Weighted_Sum + (L_Adaptive_Delta * L_Adaptive_Weight);
        L_Adaptive_Weight_Total := L_Adaptive_Weight_Total + L_Adaptive_Weight;
    END_IF;
END_FOR;

IF L_Adaptive_Weight_Total > 0.0 THEN
    L_Adaptive_Effective_Delta := L_Adaptive_Weighted_Sum / L_Adaptive_Weight_Total;
END_IF;

IF L_Adaptive_Effective_Delta > 1.5 THEN
    L_Adaptive_Correction := 2.0;
ELSIF L_Adaptive_Effective_Delta > 0.7 THEN
    L_Adaptive_Correction := 1.0;
ELSIF L_Adaptive_Effective_Delta < -1.5 THEN
    L_Adaptive_Correction := -2.0;
ELSIF L_Adaptive_Effective_Delta < -0.7 THEN
    L_Adaptive_Correction := -1.0;
ELSE
    L_Adaptive_Correction := 0.0;
END_IF;

IF L_Adaptive_Max_Delta > 2.5 AND L_Adaptive_Correction < 2.0 THEN
    L_Adaptive_Correction := 2.0;
END_IF;

L_Target_Supply_Temp := L_Target_Supply_Temp + L_Adaptive_Correction;

IF L_Target_Supply_Temp < 20.0 THEN
    L_Target_Supply_Temp := 20.0;
ELSIF L_Target_Supply_Temp > 45.0 THEN
    L_Target_Supply_Temp := 45.0;
END_IF;

// 2. Индивидуальное управление зонами отопления (ТЗ 1.1, 2.5)
FOR L_i := 1 TO GVL_CONSTANTS.C_MAX_HEATING_CIRCUITS DO
    fbFloorTempValidator[L_i](
        VI_Value := VI_Floor_Temps[L_i],
        VI_Min_Valid := -40.0,
        VI_Max_Valid := 120.0,
        VI_Fallback_Mode := 0
    );

    L_Climate_Zone_ID := VI_Zone_Configs[L_i].zone;
    IF L_Climate_Zone_ID >= 1 AND L_Climate_Zone_ID <= 16 THEN
        fbRoomTempValidator[L_Climate_Zone_ID](
        VI_Value := VI_Room_Temps[L_Climate_Zone_ID],
        VI_Min_Valid := -40.0,
        VI_Max_Valid := 120.0,
        VI_Fallback_Mode := 0
        );
    END_IF;

    // Контроль перегрева стяжки (защита напольного покрытия)
    L_Overheat_Timer[L_i](IN := fbFloorTempValidator[L_i].VO_Value > VI_Config.Overheat_Threshold, PT := T#60s, VI_System_Time_MS := VI_System_Time_MS);

    // Выбор датчика температуры с автоматическим переключением при неисправности
    L_Current_Temp := 0.0;
    L_Sensor_Error := FALSE;

    IF VI_Zone_Configs[L_i].control_type = 1 OR VI_Zone_Configs[L_i].control_type = 2 THEN
        // Основной: по воздуху
        IF NOT fbRoomTempValidator[L_Climate_Zone_ID].VO_Error THEN
            L_Current_Temp := fbRoomTempValidator[L_Climate_Zone_ID].VO_Value;
        ELSIF NOT fbFloorTempValidator[L_i].VO_Error THEN
            L_Current_Temp := fbFloorTempValidator[L_i].VO_Value; // Резервный: по полу
        ELSE
            L_Sensor_Error := TRUE;
        END_IF;
    ELSE
        // Основной: по полу
        IF NOT fbFloorTempValidator[L_i].VO_Error THEN
            L_Current_Temp := fbFloorTempValidator[L_i].VO_Value;
        ELSIF NOT fbRoomTempValidator[L_Climate_Zone_ID].VO_Error THEN
            L_Current_Temp := fbRoomTempValidator[L_Climate_Zone_ID].VO_Value; // Резервный: по воздуху
        ELSE
            L_Sensor_Error := TRUE;
        END_IF;
    END_IF;

    IF L_Sensor_Error THEN
        L_Any_Sensor_Error := TRUE;
        VO_Zone_Valves[L_i] := FALSE; // Безопасное состояние при ошибке обоих датчиков
    ELSE
        // ПИД-регулирование и ШИМ для каждой зоны
        // Применяем плавную корректировку уставки от сценария
        L_Zone_Config := VI_Zone_Configs[L_i];
        L_Zone_Config.design_temp := L_Zone_Config.design_temp + L_Scenario_Adjust;
        L_Floor_Controllers[L_i](
            VI_Current_Temp := L_Current_Temp,
            VI_Config := L_Zone_Config,
            VI_Tariff := VI_Tariff,
            VI_Current_Hour := VI_Current_Hour,
            VI_IsActivePLC := VI_IsActivePLC,
            VI_System_Time_MS := VI_System_Time_MS,
            VO_Valve_Bool => VO_Zone_Valves[L_i]
        );
    END_IF;

    // Принудительное закрытие клапана при перегреве пола (ТЗ 2.5)
    IF L_Overheat_Timer[L_i].Q THEN
        VO_Zone_Valves[L_i] := FALSE;
    END_IF;

    // Обработка действий от Rule Engine (ТЗ 13.0)
    FOR L_j := 1 TO GVL_CONSTANTS.C_MAX_RULES DO
        IF VI_Rule_Actions[L_j].Active AND VI_Rule_Actions[L_j].Target_ID = L_i THEN
            IF VI_Rule_Actions[L_j].Action_Type = E_Rule_Action_Type.ACTION_SET_FLOOR_HEATING THEN
                VO_Zone_Valves[L_i] := (VI_Rule_Actions[L_j].Value > 0.5);
            END_IF;
        END_IF;
    END_FOR;
END_FOR;

GVL_STATE.G_Heating_Sensor_Fault := L_Any_Sensor_Error;

// 3. Определение потребности в работе коллекторных насосов
FOR L_i := 1 TO GVL_CONSTANTS.C_MAX_MANIFOLDS DO
    L_Any_Zone_Active[L_i] := FALSE;
END_FOR;

FOR L_i := 1 TO GVL_CONSTANTS.C_MAX_HEATING_CIRCUITS DO
    IF VO_Zone_Valves[L_i] THEN
        L_j := VI_Zone_Configs[L_i].manifold_id;
        IF L_j >= 1 AND L_j <= GVL_CONSTANTS.C_MAX_MANIFOLDS THEN
            L_Any_Zone_Active[L_j] := TRUE;
        END_IF;
    END_IF;
END_FOR;

// 4. Управление смесительными узлами коллекторов (ТЗ 2.6, 12.2)
FOR L_i := 1 TO GVL_CONSTANTS.C_MAX_MANIFOLDS DO
    // ПИД-регулирование трехходового клапана для поддержания стабильной температуры подачи
    // Вызываем ПИД регулятор каждую секунду
    L_PID_Timer[L_i](IN := TRUE, PT := T#1s, VI_System_Time_MS := VI_System_Time_MS);
    IF L_PID_Timer[L_i].Q THEN
        L_PID_Timer[L_i](IN := FALSE, PT := T#1s, VI_System_Time_MS := VI_System_Time_MS); // Сброс таймера
        L_PID_Timer[L_i](IN := TRUE, PT := T#1s, VI_System_Time_MS := VI_System_Time_MS); // Перезапуск

        L_PID_Valves[L_i](
            VI_SetPoint := L_Target_Supply_Temp,
            VI_ProcessValue := VI_Manifold_Temps_Supply[L_i],
            VI_Kp := 2.0, VI_Tn := 120.0, VI_Tv := 0.0,
            VI_Y_Min := 0.0, VI_Y_Max := 100.0, VI_Cycle_Time_S := 1.0,
            VO_Output => VO_Manifold_Valves[L_i]
        );
    END_IF;

    // ТЗ 2.6: Реализация обязательной паузы насоса (защита от закисания и перегрева при 72ч работе)
    L_Pump_Run_Timer[L_i](IN := VO_Manifold_Pumps[L_i] AND NOT L_Pump_In_Pause[L_i], PT := T#72h, VI_System_Time_MS := VI_System_Time_MS);
    IF L_Pump_Run_Timer[L_i].Q THEN L_Pump_In_Pause[L_i] := TRUE; END_IF;

    L_Pump_Pause_Timer[L_i](IN := L_Pump_In_Pause[L_i], PT := T#1h, VI_System_Time_MS := VI_System_Time_MS);
    IF L_Pump_Pause_Timer[L_i].Q THEN L_Pump_In_Pause[L_i] := FALSE; END_IF;

    // Включение насоса при наличии запроса от зон и отсутствии сервисной паузы
    // Приоритет ГВС: если есть запрос от ГВС, отключаем насосы отопления и закрываем клапаны
    IF VI_DHW_Heating_Demand THEN
        VO_Manifold_Pumps[L_i] := FALSE;
        VO_Manifold_Valves[L_i] := 0.0; // Принудительно закрываем смесительный клапан
    ELSE
        VO_Manifold_Pumps[L_i] := VI_IsActivePLC AND L_Any_Zone_Active[L_i] AND NOT L_Pump_In_Pause[L_i];
    END_IF;

    // Защита от замерзания системы (ТЗ 2.4)
        IF L_Freeze_Mode_Active THEN
            VO_Manifold_Pumps[L_i] := TRUE;
            IF VO_Manifold_Valves[L_i] < 35.0 THEN
                VO_Manifold_Valves[L_i] := 35.0;
            END_IF;
        END_IF;

        // Сбор диагностических данных для визуализации на HMI
    VO_Status[L_i].Pump_On := VO_Manifold_Pumps[L_i];
    VO_Status[L_i].Pump_Current := VI_Manifold_Currents[L_i];
    VO_Status[L_i].Pressure := VI_Manifold_Pressures[L_i];
    VO_Status[L_i].Temp_Supply := VI_Manifold_Temps_Supply[L_i];
    VO_Status[L_i].Temp_Return := VI_Manifold_Temps_Return[L_i];
    VO_Status[L_i].Valve_Pos := VO_Manifold_Valves[L_i];

    // Предиктивная диагностика насоса
    L_Pump_Diag[L_i](
        VI_Current_Value := VI_Manifold_Currents[L_i],
        VI_Nominal_Value := 0.55, // Номинальный ток насоса по ТЗ: середина диапазона 0.3..0.8 А
        VI_Is_Running := VO_Manifold_Pumps[L_i],
        VI_Reset_Stats := FALSE,
        VI_System_Time_MS := VI_System_Time_MS,
        VIO_Health_Data := VO_Status[L_i].Health
    );

    // Автоматический контроль рабочих параметров (ток / давление / ΔT)
        IF VO_Manifold_Pumps[L_i] THEN
            L_Delta_T := VI_Manifold_Temps_Supply[L_i] - VI_Manifold_Temps_Return[L_i];

            // Контроль тока насоса:
            // Приоритет ошибок:
            // 1. Насос/ток
            // 2. Давление
            // 3. ΔT
            VO_Status[L_i].Error := FALSE;
            VO_Status[L_i].Error_ID := 0;

            IF VI_Manifold_Currents[L_i] <= 0.01 THEN
                VO_Status[L_i].Error := TRUE;
                VO_Status[L_i].Error_ID := TO_WORD(GVL_CONFIG.ERR_PUMP_NO_CURRENT);
            ELSIF VI_Manifold_Currents[L_i] < 0.3 THEN
                VO_Status[L_i].Error := TRUE;
                VO_Status[L_i].Error_ID := TO_WORD(GVL_CONFIG.ERR_PUMP_UNDERCURRENT);
            ELSIF VI_Manifold_Currents[L_i] > 1.5 THEN
                VO_Status[L_i].Error := TRUE;
                VO_Status[L_i].Error_ID := TO_WORD(GVL_CONFIG.ERR_PUMP_OVERCURRENT);
            END_IF;

            // Проверка давления в системе (норма 1.5 - 2.5 бар)
            IF (NOT VO_Status[L_i].Error) AND (VI_Manifold_Pressures[L_i] < 1.5 OR VI_Manifold_Pressures[L_i] > 2.5) THEN
                VO_Status[L_i].Error := TRUE;
                VO_Status[L_i].Error_ID := TO_WORD(GVL_CONFIG.ERR_PRESSURE_OUT_OF_RANGE);
            END_IF;

            // Проверка эффективности теплообмена (ΔT 5..10°C норма)
            IF NOT VO_Status[L_i].Error THEN
                IF L_Delta_T < 5.0 THEN
                    VO_Status[L_i].Error := TRUE;
                    VO_Status[L_i].Error_ID := TO_WORD(GVL_CONFIG.ERR_DELTA_T_LOW);
                ELSIF L_Delta_T > 10.0 THEN
                    VO_Status[L_i].Error := TRUE;
                    VO_Status[L_i].Error_ID := TO_WORD(GVL_CONFIG.ERR_DELTA_T_HIGH);
                END_IF;
            END_IF;
        END_IF;

        // ТЗ 12.2: Еженедельное тестирование запорной арматуры (предотвращение закисания)
    // Выполняется менеджером fbValveTestManager
END_FOR;

fbValveTestManager(
    VI_System_Time_MS := VI_System_Time_MS,
    VI_IsActivePLC := VI_IsActivePLC,
    VI_Valve_Currents := VI_Manifold_Currents,
    VI_Valve_End_Switches := VI_Manifold_End_Switches,
    VI_Config := VI_Valve_Test_Config
);

IF fbValveTestManager.VO_Test_Active THEN
    L_i := fbValveTestManager.VO_Current_Valve;
    IF L_i >= 1 AND L_i <= GVL_CONSTANTS.C_MAX_MANIFOLDS THEN
        IF fbValveTestManager.VO_Valve_Cmd[L_i] THEN
            VO_Manifold_Valves[L_i] := 100.0;
        ELSE
            VO_Manifold_Valves[L_i] := 0.0;
        END_IF;
        VO_Manifold_Pumps[L_i] := FALSE; // Отключаем насос при тестировании клапана
    END_IF;
END_IF;

// 5. Управление каскадом котлов (ТЗ 2.8, OpenTherm-only, без legacy mirror)
L_Demand_Power := 0.0;
FOR L_i := 1 TO GVL_CONSTANTS.C_MAX_MANIFOLDS DO
    IF VO_Manifold_Pumps[L_i] THEN
        L_Demand_Power := L_Demand_Power + VO_Manifold_Valves[L_i];
    END_IF;
END_FOR;

// В режиме антизамерзания обеспечиваем минимальный запрос тепла
IF L_Freeze_Mode_Active AND L_Demand_Power < 20.0 THEN
    L_Demand_Power := 20.0;
END_IF;

IF L_Policy_Degraded THEN
    IF L_Demand_Power > 60.0 THEN
        L_Demand_Power := 60.0;
    END_IF;
END_IF;

fbBoilerCascade(
    VI_Enable := VI_IsActivePLC AND ((L_Demand_Power > GVL_CONSTANTS.C_BOILER_CASCADE_MIN_DEMAND) OR L_Freeze_Mode_Active),
    VI_System_Time_MS := VI_System_Time_MS,
    VI_Boiler_Stop := FALSE,
    VI_DHW_Heating_Demand := VI_DHW_Heating_Demand,
    VI_DHW_Target_Temp := VI_DHW_Target_Temp,
    VI_Target_Supply_Temp := L_Target_Supply_Temp,
    VI_Demand_Power := L_Demand_Power,
    VI_Boiler_Flame_Status := VI_Boiler_Flame_Status,
    VI_Boiler_Error_Status := VI_Boiler_Error_Status,
    VI_Boiler_OT_Online := VI_Boiler_OT_Online,
    VI_Boiler_Modulation := VI_Boiler_Modulation,
    VO_Boiler_Enable => L_Boiler_Request_Enable,
    VO_Boiler_Setpoint => L_Boiler_Request_Setpoint,
    VO_Lead_Boiler => L_Lead_Boiler
);

// ========================================
// OT availability enforcement (no fallback)
// ========================================
FOR L_i := 1 TO GVL_CONSTANTS.C_MAX_BOILERS DO
    IF NOT VI_Boiler_OT_Online[L_i] OR VI_Boiler_Error_Status[L_i] THEN
        L_Boiler_Request_Enable[L_i] := FALSE;
        L_Boiler_Request_Setpoint[L_i] := 0.0;
    END_IF;
END_FOR;

fbBoilerOpenTherm(
    VI_Enable := L_Boiler_Request_Enable,
    VI_Setpoint := L_Boiler_Request_Setpoint,
    VI_OT_Online := VI_Boiler_OT_Online,
    VI_OT_Error := VI_Boiler_Error_Status,
    VO_OT_Enable => VO_Boiler_OT_Enable,
    VO_OT_Setpoint => VO_Boiler_OT_Setpoint,
    VO_OT_Command_Valid => L_Boiler_OT_Command_Valid
);

// ========================================
// Boiler status normalization
// ========================================
FOR L_i := 1 TO GVL_CONSTANTS.C_MAX_BOILERS DO
    // Базовый сброс диагностических флагов котла
    VO_Boiler_Status[L_i].Active := L_Boiler_Request_Enable[L_i];
    VO_Boiler_Status[L_i].Warning := FALSE;
    VO_Boiler_Status[L_i].Error := FALSE;

    // Приоритет причин:
    // 1. Нет канала OpenTherm
    // 2. Котёл вернул ошибку
    // 3. Есть запрос, но нет пламени
    IF NOT VI_Boiler_OT_Online[L_i] THEN
        VO_Boiler_Status[L_i].Error := TRUE;
        VO_Boiler_Status[L_i].Error_ID := TO_WORD(GVL_CONFIG.ERR_BOILER_OFFLINE);
        L_Any_Subsystem_Degraded := TRUE;
    ELSIF VI_Boiler_Error_Status[L_i] THEN
        VO_Boiler_Status[L_i].Error := TRUE;
        VO_Boiler_Status[L_i].Error_ID := TO_WORD(GVL_CONFIG.ERR_BOILER_GENERAL_FAULT);
        L_Any_Subsystem_Degraded := TRUE;
    ELSIF L_Boiler_Request_Enable[L_i] AND NOT VI_Boiler_Flame_Status[L_i] THEN
        VO_Boiler_Status[L_i].Warning := TRUE;
        VO_Boiler_Status[L_i].Error_ID := TO_WORD(GVL_CONFIG.ERR_BOILER_NO_FLAME);
        L_Any_Subsystem_Degraded := TRUE;
    ELSE
        VO_Boiler_Status[L_i].Error_ID := 0;
    END_IF;
END_FOR;

// Расчет наработки и остаточного ресурса котлов (ТЗ 2.8)
IF NOT L_Scan_Time_Init THEN
    L_Last_Scan_Time := VI_System_Time_MS;
    L_Scan_Time_Init := TRUE;
END_IF;

L_Delta_MS := (SEL(VI_System_Time_MS >= L_Last_Scan_Time, VI_System_Time_MS - L_Last_Scan_Time, (4294967295 - L_Last_Scan_Time) + VI_System_Time_MS + 1));
IF L_Delta_MS > 1000 THEN
    L_Delta_MS := 1000; // Ограничение дельты для предотвращения скачков после перезагрузки
END_IF;

L_Last_Scan_Time := VI_System_Time_MS;

FOR L_i := 1 TO GVL_CONSTANTS.C_MAX_BOILERS DO
    VO_Boiler_Status[L_i].Work_Seconds := GVL_Retain.G_Boiler_Work_Seconds[L_i];

    IF VI_Boiler_Flame_Status[L_i] THEN
        GVL_Retain.G_Boiler_Accumulated_MS[L_i] := GVL_Retain.G_Boiler_Accumulated_MS[L_i] + L_Delta_MS;
        IF GVL_Retain.G_Boiler_Accumulated_MS[L_i] >= GVL_CONSTANTS.C_MS_IN_SECOND THEN
            GVL_Retain.G_Boiler_Work_Seconds[L_i] := GVL_Retain.G_Boiler_Work_Seconds[L_i] + (GVL_Retain.G_Boiler_Accumulated_MS[L_i] / 1000);
            GVL_Retain.G_Boiler_Accumulated_MS[L_i] := GVL_Retain.G_Boiler_Accumulated_MS[L_i] MOD 1000;

            // Защита от переполнения (сброс при достижении ~136 лет)
            IF GVL_Retain.G_Boiler_Work_Seconds[L_i] > 4000000000 THEN
                GVL_Retain.G_Boiler_Work_Seconds[L_i] := 0;
            END_IF;

            VO_Boiler_Status[L_i].Work_Seconds := GVL_Retain.G_Boiler_Work_Seconds[L_i];
        END_IF;
    END_IF;

    VO_Boiler_Status[L_i].Work_Hours := TO_REAL(VO_Boiler_Status[L_i].Work_Seconds) / 3600.0;

    L_Boiler_Life[L_i](
        VI_Runtime_Hours := TO_UDINT(VO_Boiler_Status[L_i].Work_Hours),
        VI_Start_Count := 0, // Не считаем пуски для котлов в этой версии
        VI_Nominal_Life := 50000 // 50,000 часов
    );
    VO_Boiler_Status[L_i].Resource_Percent := TO_REAL(L_Boiler_Life[L_i].VO_Remaining_Percent);
    VO_Boiler_Status[L_i].Running := VI_Boiler_Flame_Status[L_i];
END_FOR;
GVL_STATE.G_Heating_Subsystem_Degraded := L_Any_Subsystem_Degraded;

END_FUNCTION_BLOCK
// >>> BULK_SYNC_ANCHOR: FB_Heating_System_Manager <<<

(* ---- FB_Rule_Engine.st ---- *)
FUNCTION_BLOCK FB_Rule_Engine
VAR_INPUT
    VI_System_Time_MS : UDINT; // Системное время (мс)
    VI_IsActivePLC : BOOL; // Флаг: Данный ПЛК является ведущим
    VI_Security_Armed : BOOL; // Статус: Система под охраной
    VI_Current_Time : TOD; // Текущее время суток
    VI_Day_Of_Week : INT; // Текущий день недели (1..7, 1 = Понедельник)
END_VAR
VAR_IN_OUT
    VI_Rules : ARRAY[1..GVL_CONSTANTS.C_MAX_RULES] OF ST_User_Rule; // Массив пользовательских правил
    VI_Indoor_Temps : ARRAY[1..16] OF REAL; // Температуры в помещениях
    VI_Floor_Temps : ARRAY[1..8] OF REAL; // Температуры пола
    VI_Humidities : ARRAY[1..16] OF REAL; // Влажность в помещениях
    VI_CO2_Levels : ARRAY[1..16] OF REAL; // Уровни CO2
    VI_Motion_Sensors : ARRAY[1..16] OF BOOL; // Датчики движения
    VI_Door_Sensors : ARRAY[1..GVL_CONSTANTS.C_MAX_DOOR_SENSORS] OF BOOL; // Датчики открытия дверей
    VI_Window_Sensors : ARRAY[1..16] OF BOOL; // Датчики открытия окон
    VI_Water_Sensors : ARRAY[1..GVL_CONSTANTS.C_MAX_FLOOD_SENSORS] OF BOOL; // Датчики протечки воды
    VI_Smoke_Sensors : ARRAY[1..GVL_CONSTANTS.C_MAX_SMOKE_SENSORS] OF BOOL; // Датчики дыма
    VI_Methane_Sensors : ARRAY[1..GVL_CONSTANTS.C_MAX_METHANE_SENSORS] OF REAL; // Датчики метана
    VI_CO_Sensors : ARRAY[1..GVL_CONSTANTS.C_MAX_CO_SENSORS] OF REAL; // Датчики угарного газа
END_VAR
VAR_OUTPUT
    VO_Preheat_Request : BOOL; // pre-departure heating trigger
    VO_Actions : ARRAY[1..GVL_CONSTANTS.C_MAX_RULES] OF ST_Rule_Action; // Сформированные действия по правилам
END_VAR
VAR
    L_i : INT;
    L_Condition_Met : BOOL;
    L_Current_Value : REAL;
    L_Triggers : ARRAY[1..GVL_CONSTANTS.C_MAX_RULES] OF R_TRIG;
    L_Trigger_Count : ARRAY[1..GVL_CONSTANTS.C_MAX_RULES] OF UINT;
    L_Last_Reset_Time : UDINT;
    L_Elapsed_Time : UDINT;
END_VAR

IF NOT VI_IsActivePLC THEN RETURN; END_IF;

VO_Preheat_Request := FALSE;

// Сброс счетчиков срабатываний каждую минуту (защита от циклических зависимостей/дребезга)
L_Elapsed_Time := (SEL(VI_System_Time_MS >= L_Last_Reset_Time, VI_System_Time_MS - L_Last_Reset_Time, (4294967295 - L_Last_Reset_Time) + VI_System_Time_MS + 1));

IF L_Elapsed_Time >= GVL_CONSTANTS.C_MS_IN_MINUTE THEN
    L_Last_Reset_Time := VI_System_Time_MS;
    FOR L_i := 1 TO GVL_CONSTANTS.C_MAX_RULES DO
        L_Trigger_Count[L_i] := 0;
    END_FOR;
END_IF;

FOR L_i := 1 TO GVL_CONSTANTS.C_MAX_RULES DO

    VO_Actions[L_i].Active := FALSE;
    IF VI_Rules[L_i].Enabled THEN
        L_Condition_Met := FALSE;
        L_Current_Value := 0.0;

        // Определение значения для проверки
        IF VI_Rules[L_i].Condition_Target_ID > 0 THEN
            CASE VI_Rules[L_i].Condition_Type OF
                E_Rule_Condition_Type.COND_AIR_TEMP: IF VI_Rules[L_i].Condition_Target_ID <= 16 THEN L_Current_Value := VI_Indoor_Temps[VI_Rules[L_i].Condition_Target_ID]; END_IF;
                E_Rule_Condition_Type.COND_FLOOR_TEMP: IF VI_Rules[L_i].Condition_Target_ID <= 8 THEN L_Current_Value := VI_Floor_Temps[VI_Rules[L_i].Condition_Target_ID]; END_IF;
                E_Rule_Condition_Type.COND_HUMIDITY: IF VI_Rules[L_i].Condition_Target_ID <= 16 THEN L_Current_Value := VI_Humidities[VI_Rules[L_i].Condition_Target_ID]; END_IF;
                E_Rule_Condition_Type.COND_CO2: IF VI_Rules[L_i].Condition_Target_ID <= 16 THEN L_Current_Value := VI_CO2_Levels[VI_Rules[L_i].Condition_Target_ID]; END_IF;
                E_Rule_Condition_Type.COND_MOTION: IF VI_Rules[L_i].Condition_Target_ID <= 16 THEN L_Current_Value := SEL(VI_Motion_Sensors[VI_Rules[L_i].Condition_Target_ID], 0.0, 1.0); END_IF;
                E_Rule_Condition_Type.COND_DOOR_WINDOW:
                    IF VI_Rules[L_i].Condition_Target_ID <= GVL_CONSTANTS.C_MAX_DOOR_SENSORS THEN
                        L_Current_Value := SEL(VI_Door_Sensors[VI_Rules[L_i].Condition_Target_ID] OR VI_Window_Sensors[VI_Rules[L_i].Condition_Target_ID], 0.0, 1.0);
                    ELSIF VI_Rules[L_i].Condition_Target_ID <= 16 THEN
                        L_Current_Value := SEL(VI_Window_Sensors[VI_Rules[L_i].Condition_Target_ID], 0.0, 1.0);
                    END_IF;
                E_Rule_Condition_Type.COND_FLOOD: IF VI_Rules[L_i].Condition_Target_ID <= GVL_CONSTANTS.C_MAX_FLOOD_SENSORS THEN L_Current_Value := SEL(VI_Water_Sensors[VI_Rules[L_i].Condition_Target_ID], 0.0, 1.0); END_IF;
                E_Rule_Condition_Type.COND_SMOKE: IF VI_Rules[L_i].Condition_Target_ID <= GVL_CONSTANTS.C_MAX_SMOKE_SENSORS THEN L_Current_Value := SEL(VI_Smoke_Sensors[VI_Rules[L_i].Condition_Target_ID], 0.0, 1.0); END_IF;
                E_Rule_Condition_Type.COND_METHANE: IF VI_Rules[L_i].Condition_Target_ID <= GVL_CONSTANTS.C_MAX_METHANE_SENSORS THEN L_Current_Value := VI_Methane_Sensors[VI_Rules[L_i].Condition_Target_ID]; END_IF;
                E_Rule_Condition_Type.COND_CO: IF VI_Rules[L_i].Condition_Target_ID <= GVL_CONSTANTS.C_MAX_CO_SENSORS THEN L_Current_Value := VI_CO_Sensors[VI_Rules[L_i].Condition_Target_ID]; END_IF;
                E_Rule_Condition_Type.COND_TIME_OF_DAY: L_Current_Value := TO_REAL(TOD_TO_UDINT(VI_Current_Time) / GVL_CONSTANTS.C_MS_IN_MINUTE); // Время в минутах
                E_Rule_Condition_Type.COND_DAY_OF_WEEK: L_Current_Value := TO_REAL(VI_Day_Of_Week);
            END_CASE;
        ELSE
            IF VI_Rules[L_i].Condition_Type = E_Rule_Condition_Type.COND_TIME_OF_DAY THEN
                L_Current_Value := TO_REAL(TOD_TO_UDINT(VI_Current_Time) / GVL_CONSTANTS.C_MS_IN_MINUTE); // Время в минутах
            ELSIF VI_Rules[L_i].Condition_Type = E_Rule_Condition_Type.COND_DAY_OF_WEEK THEN
                L_Current_Value := TO_REAL(VI_Day_Of_Week);
            END_IF;
        END_IF;

        // Проверка условия
        CASE VI_Rules[L_i].Condition_Op OF
            E_Rule_Comparison.COMP_GT: L_Condition_Met := (L_Current_Value > VI_Rules[L_i].Condition_Value);
            E_Rule_Comparison.COMP_LT: L_Condition_Met := (L_Current_Value < VI_Rules[L_i].Condition_Value);
            E_Rule_Comparison.COMP_EQ: L_Condition_Met := (ABS(L_Current_Value - VI_Rules[L_i].Condition_Value) < 0.1);
            E_Rule_Comparison.COMP_GE: L_Condition_Met := (L_Current_Value >= VI_Rules[L_i].Condition_Value);
            E_Rule_Comparison.COMP_LE: L_Condition_Met := (L_Current_Value <= VI_Rules[L_i].Condition_Value);
            E_Rule_Comparison.COMP_IN_RANGE: L_Condition_Met := (L_Current_Value >= VI_Rules[L_i].Condition_Value) AND (L_Current_Value <= VI_Rules[L_i].Condition_Value_Max);
            E_Rule_Comparison.COMP_TRUE: L_Condition_Met := (L_Current_Value > 0.5);
            E_Rule_Comparison.COMP_FALSE: L_Condition_Met := (L_Current_Value < 0.5);
        END_CASE;

        // Формирование действия
        L_Triggers[L_i](CLK := L_Condition_Met);

        IF L_Triggers[L_i].Q THEN
            L_Trigger_Count[L_i] := L_Trigger_Count[L_i] + 1;
            IF L_Trigger_Count[L_i] > 10 THEN
                // ТЗ 13.5: Блокировка правила при слишком частом срабатывании (циклическая зависимость)
                VO_Actions[L_i].Active := FALSE;
                VO_Actions[L_i].Triggered := FALSE;
                CONTINUE; // Пропускаем выполнение
            END_IF;
        END_IF;

        IF L_Condition_Met AND (L_Trigger_Count[L_i] <= 10) THEN
            VO_Actions[L_i].Active := TRUE;
            VO_Actions[L_i].Triggered := L_Triggers[L_i].Q;
            VO_Actions[L_i].Action_Type := VI_Rules[L_i].Action_Type;
            VO_Actions[L_i].Target_ID := VI_Rules[L_i].Action_Target_ID;
            VO_Actions[L_i].Value := VI_Rules[L_i].Action_Value;
        END_IF;
    END_IF;
END_FOR;
// >>> BULK_SYNC_ANCHOR: FB_Rule_Engine <<<

(* ---- FB_Scenario_Transition_Controller.st ---- *)
FUNCTION_BLOCK FB_Scenario_Transition_Controller
VAR_INPUT
    VI_System_Time : UDINT;
    VI_Start_Time  : UDINT;
    VI_Duration    : UDINT; // Длительность перехода (мс)
    VI_Start_Value : REAL;  // Начальное значение
    VI_End_Value   : REAL;  // Конечное значение
END_VAR
VAR_OUTPUT
    VO_Current_Value : REAL; // Текущее интерполированное значение
    VO_Transition_Done : BOOL; // Флаг завершения перехода
END_VAR
VAR
    L_Elapsed : UDINT;
    L_Progress : REAL;
END_VAR

L_Elapsed := (SEL(VI_System_Time >= VI_Start_Time, VI_System_Time - VI_Start_Time, (4294967295 - VI_Start_Time) + VI_System_Time + 1));

IF L_Elapsed >= VI_Duration OR VI_Duration = 0 THEN
    VO_Current_Value := VI_End_Value;
    VO_Transition_Done := TRUE;
ELSE
    L_Progress := UDINT_TO_REAL(L_Elapsed) / UDINT_TO_REAL(VI_Duration);
    VO_Current_Value := VI_Start_Value + (VI_End_Value - VI_Start_Value) * L_Progress;
    VO_Transition_Done := FALSE;
END_IF;

(* ---- FB_Security_System_Manager.st ---- *)
FUNCTION_BLOCK FB_Security_System_Manager
VAR_INPUT
    VI_System_Time_MS : UDINT; // Системное время (мс)
    VI_IsActivePLC : BOOL; // Флаг: Данный ПЛК является ведущим
    VI_Arm_Request : BOOL; // Запрос на постановку под охрану
    VI_Disarm_Request : BOOL; // Запрос на снятие с охраны
    VI_PIN_Code : STRING(4); // ПИН-код для авторизации
    VI_RFID_Tag : STRING(20); // RFID/NFC метка для авторизации
    VI_2FA_Code : STRING(6); // Код двухфакторной аутентификации
    VI_Config : ST_Security_Global_Config; // Конфигурация охранной системы
    VI_Current_TOD : TOD; // Текущее время суток (от FB_Astro_Timer)
END_VAR
VAR_IN_OUT
    VI_Motion_Sensors : ARRAY[1..16] OF BOOL; // Датчики движения
    VI_Door_Sensors : ARRAY[1..GVL_CONSTANTS.C_MAX_DOOR_SENSORS] OF BOOL; // Датчики открытия дверей (герконы)
    VI_Window_Sensors : ARRAY[1..16] OF BOOL; // Датчики открытия окон (герконы)
    VI_Bypass_Motion : ARRAY[1..16] OF BOOL; // Байпас датчиков движения
    VI_Bypass_Doors : ARRAY[1..GVL_CONSTANTS.C_MAX_DOOR_SENSORS] OF BOOL; // Байпас дверей
    VI_Bypass_Windows : ARRAY[1..16] OF BOOL; // Байпас окон
END_VAR
VAR_OUTPUT
    VO_Armed : BOOL; // Статус: Система под охраной
    VO_Alarm_Active : BOOL; // Статус: Тревога активна
    VO_Siren_Active : BOOL; // Команда: Включить сирену
    VO_Status_Msg : STRING(200); // Строковое сообщение о статусе
    VO_Send_Code_Req : BOOL; // Запрос на отправку кода 2FA
    VO_Code_To_Send : STRING(6); // Сгенерированный код 2FA для отправки
END_VAR
VAR
    L_i : INT;
    L_Any_Sensor_Active : BOOL;
    L_Arm_Delay_Timer : FB_System_Timer;
    L_Alarm_Delay_Timer : FB_System_Timer;
    L_Arming_In_Progress : BOOL;
    L_Valid_PIN : BOOL;
    fbAccessCode : FB_AccessCode_Manager;
    fbTwoFactor : FB_TwoFactor_Auth;
    L_2FA_Required : BOOL;
    L_Disarm_Pending : BOOL;
    L_Reset_2FA : BOOL;
    L_Auto_Arm_Trigger : BOOL;
    R_Trig_Auto_Arm : R_TRIG;
END_VAR

IF NOT VI_IsActivePLC THEN
    VO_Armed := FALSE;
    VO_Alarm_Active := FALSE;
    VO_Siren_Active := FALSE;
    VO_Send_Code_Req := FALSE;
    VO_Code_To_Send := '';
    VO_Status_Msg := 'Охрана: резервный ПЛК';
    L_Arming_In_Progress := FALSE;
    L_Disarm_Pending := FALSE;
    L_2FA_Required := FALSE;
    L_Reset_2FA := FALSE;
    RETURN;
END_IF;

// 1. Проверка PIN-кода или RFID-метки через менеджер кодов
fbAccessCode(
    VI_System_Time_MS := VI_System_Time_MS,
    VI_IsActivePLC := VI_IsActivePLC,
    VI_Code_To_Check := VI_PIN_Code,
    VI_RFID_To_Check := VI_RFID_Tag,
    VI_Access_Codes := GVL_RETAIN.G_Access_Codes,
    VI_RFID_Tags := GVL_RETAIN.G_RFID_Tags,
    VO_Code_Valid => L_Valid_PIN
);

// 2. Логика постановки на охрану (с задержкой на выход)
L_Auto_Arm_Trigger := FALSE;
IF VI_Config.auto_arm_enabled THEN
    IF VI_Current_TOD >= UDINT_TO_TOD(VI_Config.auto_arm_time_ms) THEN
        L_Auto_Arm_Trigger := TRUE;
    END_IF;
END_IF;
R_Trig_Auto_Arm(CLK := L_Auto_Arm_Trigger);

IF ((VI_Arm_Request AND L_Valid_PIN) OR R_Trig_Auto_Arm.Q) AND NOT VO_Armed AND NOT L_Arming_In_Progress THEN
    // Проверка, что все двери/окна закрыты перед постановкой (с учетом байпаса)
    L_Any_Sensor_Active := FALSE;
    FOR L_i := 1 TO GVL_CONSTANTS.C_MAX_DOOR_SENSORS DO IF VI_Door_Sensors[L_i] AND NOT VI_Bypass_Doors[L_i] THEN L_Any_Sensor_Active := TRUE; END_IF; END_FOR;
    FOR L_i := 1 TO 16 DO IF VI_Window_Sensors[L_i] AND NOT VI_Bypass_Windows[L_i] THEN L_Any_Sensor_Active := TRUE; END_IF; END_FOR;

    IF NOT L_Any_Sensor_Active THEN
        L_Arming_In_Progress := TRUE;
        VO_Status_Msg := 'Постановка на охрану. Покиньте помещение.';
    ELSE
        VO_Status_Msg := 'Ошибка постановки: Открыты двери или окна';
    END_IF;
END_IF;

L_Arm_Delay_Timer(IN := L_Arming_In_Progress, PT := TO_TIME(VI_Config.exit_delay_seconds * 1000), VI_System_Time_MS := VI_System_Time_MS);
IF L_Arm_Delay_Timer.Q THEN
    L_Arming_In_Progress := FALSE;
    VO_Armed := TRUE;
    VO_Status_Msg := 'Система под охраной';
END_IF;

// 3. Логика снятия с охраны с 2FA
IF VI_Disarm_Request AND L_Valid_PIN AND VO_Armed THEN
    IF VI_Config.enable_2fa THEN
        L_Disarm_Pending := TRUE;
        L_2FA_Required := TRUE;
        VO_Status_Msg := 'Ожидание 2FA для снятия с охраны';
    ELSE
        // Снятие без 2FA
        VO_Armed := FALSE;
        VO_Alarm_Active := FALSE;
        VO_Siren_Active := FALSE;
        L_Arming_In_Progress := FALSE;
        VO_Status_Msg := 'Система снята с охраны';
    END_IF;
END_IF;

fbTwoFactor(
    VI_System_Time_MS := VI_System_Time_MS,
    VI_Start_Auth := L_2FA_Required,
    VI_Method := E_TwoFactor_Method.TF_METHOD_TOTP, // Для примера
    VI_User_Code := VI_2FA_Code, // Используем отдельный вход для 2FA кода
    VI_Reset_Success := L_Reset_2FA
);

VO_Send_Code_Req := fbTwoFactor.VO_Send_Code_Req;
VO_Code_To_Send := fbTwoFactor.VO_Code_To_Send;

IF L_Disarm_Pending AND fbTwoFactor.VO_State.Is_Success THEN
    VO_Armed := FALSE;
    VO_Alarm_Active := FALSE;
    VO_Siren_Active := FALSE;
    L_Arming_In_Progress := FALSE;
    L_Disarm_Pending := FALSE;
    L_2FA_Required := FALSE;
    L_Reset_2FA := TRUE;
    VO_Status_Msg := 'Система снята с охраны';
ELSIF L_Disarm_Pending AND fbTwoFactor.VO_State.Is_Locked THEN
    L_Disarm_Pending := FALSE;
    L_2FA_Required := FALSE;
    L_Reset_2FA := FALSE;
    VO_Status_Msg := 'Ошибка 2FA: Превышено количество попыток';
ELSE
    L_Reset_2FA := FALSE;
END_IF;

// 4. Логика тревоги (с задержкой на вход)
IF VO_Armed THEN
    L_Any_Sensor_Active := FALSE;
    FOR L_i := 1 TO 16 DO IF VI_Motion_Sensors[L_i] AND NOT VI_Bypass_Motion[L_i] THEN L_Any_Sensor_Active := TRUE; END_IF; END_FOR;
    FOR L_i := 1 TO GVL_CONSTANTS.C_MAX_DOOR_SENSORS DO IF VI_Door_Sensors[L_i] AND NOT VI_Bypass_Doors[L_i] THEN L_Any_Sensor_Active := TRUE; END_IF; END_FOR;
    FOR L_i := 1 TO 16 DO IF VI_Window_Sensors[L_i] AND NOT VI_Bypass_Windows[L_i] THEN L_Any_Sensor_Active := TRUE; END_IF; END_FOR;

    // Защелкиваем факт нарушения периметра, чтобы кратковременное срабатывание датчика не сбрасывало таймер
    IF L_Any_Sensor_Active THEN
        L_Alarm_Delay_Timer.IN := TRUE;
    END_IF;

    L_Alarm_Delay_Timer(PT := TO_TIME(VI_Config.entry_delay_seconds * 1000), VI_System_Time_MS := VI_System_Time_MS);

    IF L_Alarm_Delay_Timer.Q THEN
        VO_Alarm_Active := TRUE;
        VO_Siren_Active := TRUE;
        VO_Status_Msg := 'ТРЕВОГА! Нарушение периметра';
    ELSIF L_Alarm_Delay_Timer.IN THEN
        VO_Status_Msg := 'Внимание! Введите PIN-код для отмены тревоги';
    END_IF;
ELSE
    L_Alarm_Delay_Timer(IN := FALSE, PT := T#0s, VI_System_Time_MS := VI_System_Time_MS); // Сброс таймера при снятии с охраны
END_IF;
// >>> BULK_SYNC_ANCHOR: FB_Security_System_Manager <<<

(* ---- FB_SHA1.st ---- *)
FUNCTION_BLOCK FB_SHA1
VAR_INPUT
    Length : INT;
END_VAR
VAR_IN_OUT
    Data : ARRAY[0..127] OF BYTE;
END_VAR
VAR_OUTPUT
    Hash : ARRAY[0..19] OF BYTE;
END_VAR
VAR
    H0, H1, H2, H3, H4 : DWORD;
    A, B, C, D, E, F, K, Temp : DWORD;
    W : ARRAY[0..79] OF DWORD;
    i, j, t : INT;
    PaddedData : ARRAY[0..127] OF BYTE;
    PaddedLength : INT;
    NumBlocks : INT;
    BlockOffset : INT;
END_VAR

// Initialize variables
H0 := 16#67452301;
H1 := 16#EFCDAB89;
H2 := 16#98BADCFE;
H3 := 16#10325476;
H4 := 16#C3D2E1F0;

// Pre-processing
FOR i := 0 TO Length - 1 DO
    PaddedData[i] := Data[i];
END_FOR;

// Append the bit '1' to the message
PaddedData[Length] := 16#80;

// Append 0 <= k < 512 bits '0', such that the resulting message length in bits
// is congruent to -64 ≡ 448 (mod 512)
PaddedLength := Length + 1;
WHILE (PaddedLength MOD 64) <> 56 DO
    PaddedData[PaddedLength] := 0;
    PaddedLength := PaddedLength + 1;
END_WHILE;

// Append length of message (before pre-processing), in bits, as 64-bit big-endian integer
// Since our message is small (max 127 bytes), we only need the lower 32 bits
Temp := TO_DWORD(Length * 8);
PaddedData[PaddedLength] := 0;
PaddedData[PaddedLength+1] := 0;
PaddedData[PaddedLength+2] := 0;
PaddedData[PaddedLength+3] := 0;
PaddedData[PaddedLength+4] := TO_BYTE(SHR(Temp, 24));
PaddedData[PaddedLength+5] := TO_BYTE(SHR(Temp, 16));
PaddedData[PaddedLength+6] := TO_BYTE(SHR(Temp, 8));
PaddedData[PaddedLength+7] := TO_BYTE(Temp);
PaddedLength := PaddedLength + 8;

NumBlocks := PaddedLength / 64;

// Process the message in successive 512-bit chunks
FOR i := 0 TO NumBlocks - 1 DO
    BlockOffset := i * 64;

    // Break chunk into sixteen 32-bit big-endian words w[i], 0 <= i <= 15
    FOR j := 0 TO 15 DO
        W[j] := SHL(TO_DWORD(PaddedData[BlockOffset + j*4]), 24) OR
                SHL(TO_DWORD(PaddedData[BlockOffset + j*4 + 1]), 16) OR
                SHL(TO_DWORD(PaddedData[BlockOffset + j*4 + 2]), 8) OR
                TO_DWORD(PaddedData[BlockOffset + j*4 + 3]);
    END_FOR;

    // Message schedule: extend the sixteen 32-bit words into eighty 32-bit words
    FOR j := 16 TO 79 DO
        Temp := W[j-3] XOR W[j-8] XOR W[j-14] XOR W[j-16];
        W[j] := SHL(Temp, 1) OR SHR(Temp, 31); // Left rotate by 1
    END_FOR;

    // Initialize hash value for this chunk
    A := H0;
    B := H1;
    C := H2;
    D := H3;
    E := H4;

    // Main loop
    FOR j := 0 TO 79 DO
        IF j <= 19 THEN
            F := (B AND C) OR ((NOT B) AND D);
            K := 16#5A827999;
        ELSIF j <= 39 THEN
            F := B XOR C XOR D;
            K := 16#6ED9EBA1;
        ELSIF j <= 59 THEN
            F := (B AND C) OR (B AND D) OR (C AND D);
            K := 16#8F1BBCDC;
        ELSE
            F := B XOR C XOR D;
            K := 16#CA62C1D6;
        END_IF;

        Temp := (SHL(A, 5) OR SHR(A, 27)) + F + E + K + W[j];
        E := D;
        D := C;
        C := SHL(B, 30) OR SHR(B, 2);
        B := A;
        A := Temp;
    END_FOR;

    // Add this chunk's hash to result so far
    H0 := H0 + A;
    H1 := H1 + B;
    H2 := H2 + C;
    H3 := H3 + D;
    H4 := H4 + E;
END_FOR;

// Produce the final hash value (big-endian)
Hash[0] := TO_BYTE(SHR(H0, 24)); Hash[1] := TO_BYTE(SHR(H0, 16)); Hash[2] := TO_BYTE(SHR(H0, 8)); Hash[3] := TO_BYTE(H0);
Hash[4] := TO_BYTE(SHR(H1, 24)); Hash[5] := TO_BYTE(SHR(H1, 16)); Hash[6] := TO_BYTE(SHR(H1, 8)); Hash[7] := TO_BYTE(H1);
Hash[8] := TO_BYTE(SHR(H2, 24)); Hash[9] := TO_BYTE(SHR(H2, 16)); Hash[10] := TO_BYTE(SHR(H2, 8)); Hash[11] := TO_BYTE(H2);
Hash[12] := TO_BYTE(SHR(H3, 24)); Hash[13] := TO_BYTE(SHR(H3, 16)); Hash[14] := TO_BYTE(SHR(H3, 8)); Hash[15] := TO_BYTE(H3);
Hash[16] := TO_BYTE(SHR(H4, 24)); Hash[17] := TO_BYTE(SHR(H4, 16)); Hash[18] := TO_BYTE(SHR(H4, 8)); Hash[19] := TO_BYTE(H4);

(* ---- PRG_Command_Verifier.st ---- *)
PROGRAM PRG_Command_Verifier
VAR
    L_Mismatch_Count : INT := 0;
END_VAR

L_Mismatch_Count := 0;

IF GVL_COMMAND.G_Gas_Valve_Close <> GVL_COMMAND_SHADOW.G_Gas_Valve_Close THEN
    L_Mismatch_Count := L_Mismatch_Count + 1;
END_IF;

IF GVL_COMMAND.G_Boiler_Stop <> GVL_COMMAND_SHADOW.G_Boiler_Stop THEN
    L_Mismatch_Count := L_Mismatch_Count + 1;
END_IF;

IF GVL_COMMAND.G_Vent_Stop <> GVL_COMMAND_SHADOW.G_Vent_Stop THEN
    L_Mismatch_Count := L_Mismatch_Count + 1;
END_IF;

IF GVL_COMMAND.G_Supply_100_Req <> GVL_COMMAND_SHADOW.G_Supply_100_Req THEN
    L_Mismatch_Count := L_Mismatch_Count + 1;
END_IF;

IF GVL_COMMAND.G_Supply_80_Req <> GVL_COMMAND_SHADOW.G_Supply_80_Req THEN
    L_Mismatch_Count := L_Mismatch_Count + 1;
END_IF;

IF GVL_COMMAND.G_Vent_PV3_Boost <> GVL_COMMAND_SHADOW.G_Vent_PV3_Boost THEN
    L_Mismatch_Count := L_Mismatch_Count + 1;
END_IF;

IF GVL_COMMAND.G_Close_Valve_35 <> GVL_COMMAND_SHADOW.G_Close_Valve_35 THEN
    L_Mismatch_Count := L_Mismatch_Count + 1;
END_IF;

IF GVL_COMMAND.G_Close_Valve_36 <> GVL_COMMAND_SHADOW.G_Close_Valve_36 THEN
    L_Mismatch_Count := L_Mismatch_Count + 1;
END_IF;

IF GVL_COMMAND.G_Lock_1_Open <> GVL_COMMAND_SHADOW.G_Lock_1_Open THEN
    L_Mismatch_Count := L_Mismatch_Count + 1;
END_IF;

IF GVL_COMMAND.G_Lock_1_Close <> GVL_COMMAND_SHADOW.G_Lock_1_Close THEN
    L_Mismatch_Count := L_Mismatch_Count + 1;
END_IF;

IF GVL_COMMAND.G_Lock_2_Open <> GVL_COMMAND_SHADOW.G_Lock_2_Open THEN
    L_Mismatch_Count := L_Mismatch_Count + 1;
END_IF;

IF GVL_COMMAND.G_Lock_2_Close <> GVL_COMMAND_SHADOW.G_Lock_2_Close THEN
    L_Mismatch_Count := L_Mismatch_Count + 1;
END_IF;

// NEW: gate/wicket verification
IF GVL_COMMAND.G_Gate_Open <> GVL_COMMAND_SHADOW.G_Gate_Open THEN
    L_Mismatch_Count := L_Mismatch_Count + 1;
END_IF;

IF GVL_COMMAND.G_Wicket_Open <> GVL_COMMAND_SHADOW.G_Wicket_Open THEN
    L_Mismatch_Count := L_Mismatch_Count + 1;
END_IF;

GVL_COMMAND_VERIFY.Command_Mismatch_Count := L_Mismatch_Count;
GVL_COMMAND_VERIFY.Command_Match_OK := (L_Mismatch_Count = 0);

IF L_Mismatch_Count > 0 THEN
    GVL_COMMAND_VERIFY.Command_Mismatch_Active := TRUE;
END_IF;
